# B&R Automation Studio project vibratorControlWithCurrentController (part 5)

#### brdkREST_func.c - Internal functions for library.
```c
#include <brdkREST_func.h>

unsigned short getMethod(brdk_rest_method_typ method) {
	switch(method) {
		case BRDK_REST_GET: return httpMETHOD_GET;
		case BRDK_REST_POST: return httpMETHOD_POST;
		case BRDK_REST_PUT: return httpMETHOD_PUT;
		case BRDK_REST_DELETE: return httpMETHOD_DELETE;
	}
	return httpMETHOD_GET;
}

brdk_rest_method_typ setMethod(unsigned short method) {
	switch(method) {
		case httpMETHOD_GET: return BRDK_REST_GET;
		case httpMETHOD_POST: return BRDK_REST_POST;
		case httpMETHOD_PUT: return BRDK_REST_PUT;
		case httpMETHOD_DELETE: return BRDK_REST_DELETE;
	}
	return BRDK_REST_GET;
}

void setHttpStatus(brdk_rest_response_action_typ status, unsigned long pStr) {
	switch(status) {
		case BRDK_REST_200_OK: brdkStrCpy(pStr, (unsigned long)&"200 OK"); break;
		case BRDK_REST_401_UNAUTHORIZED: brdkStrCpy(pStr, (unsigned long)&"401 Unauthorized"); break;
		case BRDK_REST_403_FORBIDDEN: brdkStrCpy(pStr, (unsigned long)&"403 Forbidden"); break;
		case BRDK_REST_404_NOT_FOUND: brdkStrCpy(pStr, (unsigned long)&"404 Not Found"); break;
		case BRDK_REST_500_INT_SERVER_ERROR: brdkStrCpy(pStr, (unsigned long)&"500 Internal Server Error"); break;
		case BRDK_REST_501_NOT_IMPLEMENTED: brdkStrCpy(pStr, (unsigned long)&"501 Not Implemented"); break;
		case BRDK_REST_503_SRV_UNAVAILABLE: brdkStrCpy(pStr, (unsigned long)&"503 Service Unavailable"); break;
		default: brdkStrCpy(pStr, (unsigned long)&"400 Bad Request"); break;
	}
}

brdk_rest_content_typ findContentType(unsigned long pStr) {
	if(brdkStrSearch(pStr, (unsigned long)&"html") > -1) return BRDK_REST_HTML;
	else if(brdkStrSearch(pStr, (unsigned long)&"plain") > -1) return BRDK_REST_TEXT;
	else if(brdkStrSearch(pStr, (unsigned long)&"json") > -1) return BRDK_REST_JSON;
	else if(brdkStrSearch(pStr, (unsigned long)&"xml") > -1) return BRDK_REST_XML;
	else if(brdkStrSearch(pStr, (unsigned long)&"csv") > -1) return BRDK_REST_CSV;
	else if(brdkStrSearch(pStr, (unsigned long)&"css") > -1) return BRDK_REST_CSS;
	else if(brdkStrSearch(pStr, (unsigned long)&"java") > -1) return BRDK_REST_JAVASCRIPT;
	else if(brdkStrSearch(pStr, (unsigned long)&"jpeg") > -1) return BRDK_REST_JPEG;
	else if(brdkStrSearch(pStr, (unsigned long)&"gzip") > -1) return BRDK_REST_GZIP;
	else if(brdkStrSearch(pStr, (unsigned long)&"zip") > -1) return BRDK_REST_ZIP;
	else if(brdkStrSearch(pStr, (unsigned long)&"png") > -1) return BRDK_REST_PNG;
	else if(brdkStrSearch(pStr, (unsigned long)&"gif") > -1) return BRDK_REST_GIF;
	else if(brdkStrSearch(pStr, (unsigned long)&"bmp") > -1) return BRDK_REST_BMP;
	else if(brdkStrSearch(pStr, (unsigned long)&"jpg") > -1) return BRDK_REST_JPG;
	return BRDK_REST_NONE;
}

void setContentType(unsigned long pDestination, brdk_rest_content_typ type) {
	switch(type) {
		case BRDK_REST_NONE: brdkStrCpy(pDestination,(unsigned long)&""); break;
		case BRDK_REST_HTML: brdkStrCpy(pDestination,(unsigned long)&"text/html"); break;
		case BRDK_REST_TEXT: brdkStrCpy(pDestination,(unsigned long)&"text/plain"); break;
		case BRDK_REST_JSON: brdkStrCpy(pDestination,(unsigned long)&"application/json"); break;
		case BRDK_REST_XML: brdkStrCpy(pDestination,(unsigned long)&"application/xml"); break;
		case BRDK_REST_CSV: brdkStrCpy(pDestination,(unsigned long)&"text/csv"); break;
		case BRDK_REST_CSS: brdkStrCpy(pDestination,(unsigned long)&"text/css"); break;
		case BRDK_REST_JAVASCRIPT: brdkStrCpy(pDestination,(unsigned long)&"text/javascript"); break;
		case BRDK_REST_JPEG: brdkStrCpy(pDestination,(unsigned long)&"image/jpeg"); break;
		case BRDK_REST_GZIP: brdkStrCpy(pDestination,(unsigned long)&"application/gzip"); break;
		case BRDK_REST_ZIP: brdkStrCpy(pDestination,(unsigned long)&"application/zip"); break;
		case BRDK_REST_PNG: brdkStrCpy(pDestination,(unsigned long)&"image/png"); break;
		case BRDK_REST_GIF: brdkStrCpy(pDestination,(unsigned long)&"image/gif"); break;
		case BRDK_REST_BMP: brdkStrCpy(pDestination,(unsigned long)&"image/bmp"); break;
		case BRDK_REST_JPG: brdkStrCpy(pDestination,(unsigned long)&"image/jpg"); break;
	}
}

unsigned char validateServerParams(brdkRESTServer_typ* inst, brdk_rest_server_internal_typ* this) {
	unsigned char i,j,validate = true;
	brdkStrCat((unsigned long)&this->uri, (unsigned long)&"&");
	for(i=0; i <= BRDK_REST_PARAMS_MAX_SIZE; i++) {
		/* try to find in uri */
		if(inst->parameters[i].pKey != 0) {
			validate = false;
			switch(inst->parameters[i].from) {

				case BRDK_REST_PARAMETERS:
					validate = brdkStrSubStrSearch(inst->parameters[i].pValue,(unsigned long)&this->uri,inst->parameters[i].pKey,(unsigned long)&("&"), 1, true);
					break;

				case BRDK_REST_HEADER:
					for(j=0; j <= BRDK_REST_PARAMS_MAX_SIZE; j++) {
						if(brdkStrCmp(inst->parameters[i].pKey, (unsigned long)&this->httpRequestHeader.userLine[j].name) == 0) {
							validate = !brdkStrIsEmpty((unsigned long)&this->httpRequestHeader.userLine[j].value);
							if(validate) {
								brdkStrCpy(inst->parameters[i].pValue, (unsigned long)&this->httpRequestHeader.userLine[j].value);
								break;
							}
						}
					}
					break;

				case BRDK_REST_BODY_JSON:
					switch(inst->parameters[i].datatype) {

						case BRDK_JSON_STRING_TO_STRING: case BRDK_JSON_DINT_TO_STRING: case BRDK_JSON_UDINT_TO_STRING: case BRDK_JSON_BOOL_TO_STRING:
							if(brdkJSONparseToString(inst->pRequestBody, inst->parameters[i].pKey, inst->parameters[i].pValue, inst->parameters[i].datatype, inst->requestBodyMaxLength, 0) > -1) {
								validate = true;
							}
							break;

						default:
							if(brdkJSONparse(inst->pRequestBody, inst->parameters[i].pKey, inst->parameters[i].pValue , inst->parameters[i].datatype, 0) > -1) {
								validate = true;
							}
							break;

					}
					break;

			}
			if(!validate) break;

		}
		else break;
	}
	return validate;
}
```

- CHANGELOG (not shown)

### Library Logical/Libraries/brdkJSON (ANSIC, version 1.00.0) - JSON handling library.
Depends on: brdkSTR

#### brdkJSON.typ - Exported data types
```iecst
TYPE
	brdk_json_find_typ :
		( (*JSON find type.*)
		BRDK_JSON_OBJECT_START := 0, (*JSON object start {.*)
		BRDK_JSON_OBJECT_END := 1, (*JSON object end }.*)
		BRDK_JSON_ARRAY_START := 2, (*JSON array start [.*)
		BRDK_JSON_ARRAY_ELEMENT := 4, (*JSON array element ,.*)
		BRDK_JSON_ARRAY_END := 5, (*JSON array end ].*)
		BRDK_JSON_OBJECT_VALUE := 6, (*JSON value :.*)
		BRDK_JSON_SOURCE_END := 7 (*JSON source end NULL.*)
		);
	brdk_json_dt_typ :
		( (*JSON datatype.*)
		BRDK_JSON_STRING_TO_STRING := 0, (*STRING -> STRING.*)
		BRDK_JSON_STRING_TO_DINT := 1, (*STRING -> DINT.*)
		BRDK_JSON_STRING_TO_UDINT := 2, (*STRING -> UDINT.*)
		BRDK_JSON_STRING_TO_REAL := 3, (*STRING -> REAL.*)
		BRDK_JSON_STRING_TO_BOOL := 4, (*STRING -> BOOL.*)
		BRDK_JSON_DINT_TO_STRING := 5, (*DINT -> STRING.*)
		BRDK_JSON_DINT_TO_DINT := 6, (*DINT -> DINT.*)
		BRDK_JSON_DINT_TO_BOOL := 7, (*DINT -> BOOL.*)
		BRDK_JSON_UDINT_TO_STRING := 8, (*UDINT -> STRING.*)
		BRDK_JSON_UDINT_TO_UDINT := 9, (*UDINT -> UDINT.*)
		BRDK_JSON_UDINT_TO_BOOL := 10, (*UDINT -> BOOL.*)
		BRDK_JSON_BOOL_TO_STRING := 11, (*BOOL -> STRING.*)
		BRDK_JSON_BOOL_TO_DINT := 12, (*BOOL -> DINT.*)
		BRDK_JSON_BOOL_TO_UDINT := 13, (*BOOL -> UDINT.*)
		BRDK_JSON_BOOL_TO_BOOL := 14, (*BOOL -> BOOL.*)
		BRDK_JSON_REAL_TO_REAL := 15, (*REAL -> REAL.*)
		BRDK_JSON_REAL_TO_STRING := 16 (*REAL -> STRING.*)
		);
END_TYPE
```

#### brdkJSON.fun - Exported functions and function blocks
```iecst
FUNCTION brdkJSONfindNext : DINT (*Find a JSON element. $RETURN=position;Position after the found element.*) (*$GROUP=User,$CAT=User,$GROUPICON=User.png,$CATICON=User.png*)
	VAR_INPUT
		pSource : UDINT := 0; (*String pointer to the source string.*)
		find : brdk_json_find_typ := BRDK_JSON_OBJECT_START; (*JSON element to find.*)
		position : UDINT := 0; (*Position in the source string where to starte the search for the element. 0 will start from the beginning.*)
	END_VAR
END_FUNCTION

FUNCTION brdkJSONnextElement : brdk_json_find_typ (*Return the next found JSON element. $RETURN=type;JSON element type.*) (*$GROUP=User,$CAT=User,$GROUPICON=User.png,$CATICON=User.png*)
	VAR_INPUT
		pSource : UDINT := 0; (*String pointer to the source string.*)
		pPposition : UDINT := 0; (*Pointer to the position in the source string where to starte the search for the element. 0 will start from the beginning.*)
	END_VAR
END_FUNCTION

FUNCTION brdkJSONparse : DINT (*Finds a name and value pair in a JSON object. $RETURN=position;Position after the found object. Can be used as position input to search for more values in a source string. See error codes below.*) (*$GROUP=User,$CAT=User,$GROUPICON=User.png,$CATICON=User.png*)
	VAR_INPUT
		pSource : UDINT := 0; (*String pointer to the source string.*)
		pName : UDINT := 0; (*String pointer to the name.*)
		pValue : UDINT := 0; (*String pointer to the value destination.*)
		datatype : brdk_json_dt_typ := BRDK_JSON_DINT_TO_DINT; (*Convert datatype.*)
		position : UDINT := 0; (*Position in the source string where to starte the search for the value. 0 will start from the beginning.*)
	END_VAR
END_FUNCTION

FUNCTION brdkJSONparseArray : DINT (*Finds a name and value pair in a JSON object. $RETURN=position;Position after the found object. Can be used as position input to search for more values in a source string. See error codes below.*) (*$GROUP=User,$CAT=User,$GROUPICON=User.png,$CATICON=User.png*)
	VAR_INPUT
		pSource : UDINT := 0; (*String pointer to the source string.*)
		pName : UDINT := 0; (*String pointer to the name.*)
		pValue : UDINT := 0; (*String pointer to the value destination.*)
		datatype : brdk_json_dt_typ := BRDK_JSON_DINT_TO_DINT; (*Convert datatype.*)
		arraySize : UDINT := 0; (*Maximum size of array (number of elements).*)
		position : UDINT := 0; (*Position in the source string where to starte the search for the value. 0 will start from the beginning.*)
	END_VAR
END_FUNCTION

FUNCTION brdkJSONparseToString : DINT (*Finds a name and value pair in a JSON object. $RETURN=position;Position after the found object. Can be used as position input to search for more values in a source string. See error codes below.*) (*$GROUP=User,$CAT=User,$GROUPICON=User.png,$CATICON=User.png*)
	VAR_INPUT
		pSource : UDINT := 0; (*String pointer to the source string.*)
		pName : UDINT := 0; (*String pointer to the name.*)
		pValue : UDINT := 0; (*String pointer to the value destination.*)
		datatype : brdk_json_dt_typ := BRDK_JSON_STRING_TO_STRING; (*Convert datatype.*)
		size : UDINT := 0; (*Maximum size of the value. Only used when value is a STRING type.*)
		position : UDINT := 0; (*Position in the source string where to starte the search for the value. 0 will start from the beginning.*)
	END_VAR
END_FUNCTION

FUNCTION brdkJSONparseToStringArray : DINT (*Finds a name and value pair in a JSON object. $RETURN=position;Position after the found object. Can be used as position input to search for more values in a source string. See error codes below.*) (*$GROUP=User,$CAT=User,$GROUPICON=User.png,$CATICON=User.png*)
	VAR_INPUT
		pSource : UDINT := 0; (*String pointer to the source string.*)
		pName : UDINT := 0; (*String pointer to the name.*)
		pValue : UDINT := 0; (*String pointer to the value destination.*)
		datatype : brdk_json_dt_typ := BRDK_JSON_STRING_TO_STRING; (*Convert datatype.*)
		size : UDINT := 0; (*Maximum size of the value. Only used when value is a STRING type.*)
		arraySize : UDINT := 0; (*Maximum size of array (number of elements).*)
		position : UDINT := 0; (*Position in the source string where to starte the search for the value. 0 will start from the beginning.*)
	END_VAR
END_FUNCTION

FUNCTION brdkJSONstringify : UDINT (*Add name and value pair to a JSON object. $RETURN=position;Position after the added object. Can be used as position input to search for more values in a source string. See error codes below.*) (*$GROUP=User,$CAT=User,$GROUPICON=User.png,$CATICON=User.png*)
	VAR_INPUT
		pDestination : UDINT := 0; (*String pointer to the destination string.*)
		pName : UDINT := 0; (*String pointer to the name.*)
		pValue : UDINT := 0; (*String pointer to value.*)
		datatype : brdk_json_dt_typ := BRDK_JSON_STRING_TO_STRING; (*Convert datatype.*)
		size : UDINT := 0; (*Maximum size of the destination STRING.*)
		position : UDINT := 0; (*Position in the source string where to starte the search for the value. 0 will start from the beginning or it will search for a }.*)
	END_VAR
END_FUNCTION
```

#### brdkJSONfindNext.c - brdkJSONfindNext implementation.
```c
#include <brdkJSON_func.h>

signed long brdkJSONfindNext(unsigned long pSource, enum brdk_json_find_typ find, unsigned long position) {
	unsigned char findChar;
	switch(find) {
		case BRDK_JSON_OBJECT_START: findChar = BRDK_STR_ASCII_OPEN_BRACE; break;
		case BRDK_JSON_OBJECT_END: findChar = BRDK_STR_ASCII_CLOSE_BRACE; break;
		case BRDK_JSON_ARRAY_START: findChar = BRDK_STR_ASCII_OPEN_BRACKET; break;
		case BRDK_JSON_ARRAY_ELEMENT: findChar = BRDK_STR_ASCII_COMMA; break;
		case BRDK_JSON_ARRAY_END: findChar = BRDK_STR_ASCII_CLOSE_BRACKET; break;
		case BRDK_JSON_OBJECT_VALUE: findChar = BRDK_STR_ASCII_COMMA; break;
		case BRDK_JSON_SOURCE_END: findChar = BRDK_STR_ASCII_NULL; break;
	}
	while(((char*)pSource)[position] != BRDK_STR_ASCII_NULL) {
		if(((char*)pSource)[position++] == findChar) {
			if(((char*)pSource)[position] != BRDK_STR_ASCII_NULL) return position;
			else return -2;
		}
	}
	return -1;
}
```

#### brdkJSONnextElement.c - brdkJSONfindNext implementation.
```c
#include <brdkJSON_func.h>

enum brdk_json_find_typ brdkJSONnextElement(unsigned long pSource, unsigned long pPosition) {
	enum brdk_json_find_typ find = BRDK_JSON_SOURCE_END;
	signed long* pos = (signed long*)pPosition;
	unsigned char run = true;
	while(run) {
		switch(((char*)pSource)[*pos]) {
			case BRDK_STR_ASCII_NULL: find = BRDK_JSON_SOURCE_END; run = false; break;
			case BRDK_STR_ASCII_OPEN_BRACE: find = BRDK_JSON_OBJECT_START; run = false; break;
			case BRDK_STR_ASCII_CLOSE_BRACE: find = BRDK_JSON_OBJECT_END; run = false; break;
			case BRDK_STR_ASCII_OPEN_BRACKET: find = BRDK_JSON_ARRAY_START; run = false; break;
			case BRDK_STR_ASCII_COMMA: find = BRDK_JSON_ARRAY_ELEMENT; run = false; break;
			case BRDK_STR_ASCII_CLOSE_BRACKET: find = BRDK_JSON_ARRAY_END; run = false; break;
			case BRDK_STR_ASCII_COLON: find = BRDK_JSON_OBJECT_VALUE; run = false; break;
			default: *pos += 1; break;
		}

	}
	*pos += 1;
	if(((char*)pSource)[*pos] == BRDK_STR_ASCII_NULL) *pos = -1;
	return find;
}
```

#### brdkJSONparse.c - brdkJSONparse implementation.
```c
#include <brdkJSON_func.h>

signed long brdkJSONparse(unsigned long pSource, unsigned long pName, unsigned long pValue, enum brdk_json_dt_typ datatype, unsigned long position) {
	/* {"test": "1234", "test2": "9876"} */
	/* {"test": 1234, "test": 9876} */
	char str[12], run, quoteCnt = 0;
	signed long i, pos = brdkStrSearch((unsigned long)&(((char*)pSource)[position]), pName);
	if(pos > -1) {
		pos += brdkStrLen(pName) + 2 + position;
		switch(datatype) {

			case BRDK_JSON_DINT_TO_DINT: case BRDK_JSON_STRING_TO_DINT:
			case BRDK_JSON_UDINT_TO_UDINT: case BRDK_JSON_STRING_TO_UDINT:
			case BRDK_JSON_REAL_TO_REAL: case BRDK_JSON_STRING_TO_REAL:
				i = 0;
				run = true;
				while(run) {
					switch(((char*)pSource)[pos]) {
						case BRDK_STR_ASCII_NULL: run = false; pos = -2; break;	/* error null cannot be here */
						case BRDK_STR_ASCII_TAB: case BRDK_STR_ASCII_SPACE: case BRDK_STR_ASCII_COLON: case BRDK_STR_ASCII_CR: case BRDK_STR_ASCII_LF: pos++; break;	/* white space and colon can be ok from beginning */
						case BRDK_STR_ASCII_COMMA: case BRDK_STR_ASCII_CLOSE_BRACE: pos++; run = false; break; /* , or } we are finished */
						case BRDK_STR_ASCII_DOUBLE_QUOTES:
							if(quoteCnt > 1 || datatype == BRDK_JSON_DINT_TO_DINT || datatype == BRDK_JSON_UDINT_TO_UDINT || datatype == BRDK_JSON_REAL_TO_REAL) {
								run = false;
								pos = -3;	/* error illegal character */
							}
							else quoteCnt++;
							pos++;
							break;
						case BRDK_STR_ASCII_HYPHEN:
							if(datatype != BRDK_JSON_DINT_TO_DINT && datatype != BRDK_JSON_STRING_TO_DINT && datatype != BRDK_JSON_REAL_TO_REAL && datatype != BRDK_JSON_STRING_TO_REAL) {
								run = false;
								pos = -3;/* error illegal character */
							}
							else ((char*)str)[i++] = ((char*)pSource)[pos++];
							break;
						case BRDK_STR_ASCII_DOT:
							if(datatype != BRDK_JSON_REAL_TO_REAL && datatype != BRDK_JSON_STRING_TO_REAL) {
								run = false;
								pos = -3;/* error illegal character */
							}
							else ((char*)str)[i++] = ((char*)pSource)[pos++];
							break;
						case BRDK_STR_ASCII_0: case BRDK_STR_ASCII_1: case BRDK_STR_ASCII_2: case BRDK_STR_ASCII_3:
						case BRDK_STR_ASCII_4: case BRDK_STR_ASCII_5: case BRDK_STR_ASCII_6: case BRDK_STR_ASCII_7:
						case BRDK_STR_ASCII_8: case BRDK_STR_ASCII_9:
							((char*)str)[i++] = ((char*)pSource)[pos++];
							break;
						default: run = false; pos = -3; break;	/* error illegal character */
					}
				}
				if(pos > -1) {
					((char*)str)[i] = BRDK_STR_ASCII_NULL;
					setValue(datatype, pValue, (unsigned long)&str);
				}
				break;

			case BRDK_JSON_BOOL_TO_BOOL: case BRDK_JSON_STRING_TO_BOOL: case BRDK_JSON_UDINT_TO_BOOL:
			case BRDK_JSON_DINT_TO_BOOL: case BRDK_JSON_BOOL_TO_DINT: case BRDK_JSON_BOOL_TO_UDINT:
				i = 0;
				run = true;
				while(run) {
					switch(((char*)pSource)[pos]) {
						case BRDK_STR_ASCII_NULL: run = false; pos = -2; break;	/* error null cannot be here */
						case BRDK_STR_ASCII_TAB: case BRDK_STR_ASCII_CR: case BRDK_STR_ASCII_LF: case BRDK_STR_ASCII_SPACE: case BRDK_STR_ASCII_COLON: pos++; break;	/* white space can be ok from beginning */
						case BRDK_STR_ASCII_DOUBLE_QUOTES:
							if(quoteCnt > 1 || datatype == BRDK_JSON_BOOL_TO_BOOL || datatype == BRDK_JSON_DINT_TO_BOOL ||
								datatype == BRDK_JSON_UDINT_TO_BOOL || datatype == BRDK_JSON_BOOL_TO_DINT || datatype == BRDK_JSON_BOOL_TO_UDINT) {
								run = false;
								pos = -3;	/* error illegal character */
							}
							else quoteCnt++;
							pos++;
							break;
						case BRDK_STR_ASCII_COMMA: case BRDK_STR_ASCII_CLOSE_BRACE: pos++; run = false; break; /* , or } we are finished */
						case BRDK_STR_ASCII_t: case BRDK_STR_ASCII_r: case BRDK_STR_ASCII_u: case BRDK_STR_ASCII_e:
						case BRDK_STR_ASCII_f: case BRDK_STR_ASCII_a: case BRDK_STR_ASCII_l: case BRDK_STR_ASCII_s:
							if(datatype != BRDK_JSON_UDINT_TO_BOOL && datatype != BRDK_JSON_DINT_TO_BOOL) ((char*)str)[i++] = ((char*)pSource)[pos++];
							else {
								run = false;
								pos = -3;	/* error illegal character */
							}
							break;

						case BRDK_STR_ASCII_0: case BRDK_STR_ASCII_1:
							((char*)str)[i++] = ((char*)pSource)[pos++];
							break;
						default: run = false; pos = -3; break;	/* error illegal character */
					}
				}
				if(pos > -1) {
					((char*)str)[i] = BRDK_STR_ASCII_NULL;
					if(datatype == BRDK_JSON_BOOL_TO_DINT) {
						signed long* tmpVal = ((signed long*)pValue);
						if(brdkStrCmp((unsigned long)&str, (unsigned long)&"true") == 0) *tmpVal = true;
						else if(brdkStrCmp((unsigned long)&str, (unsigned long)&"false") == 0) *tmpVal = false;
						else pos = -3; break;	/* error illegal character */
					}
					else if(datatype == BRDK_JSON_BOOL_TO_UDINT) {
						unsigned long* tmpVal = ((unsigned long*)pValue);
						if(brdkStrCmp((unsigned long)&str, (unsigned long)&"true") == 0) *tmpVal = true;
						else if(brdkStrCmp((unsigned long)&str, (unsigned long)&"false") == 0) *tmpVal = false;
						else pos = -3; break;	/* error illegal character */
					}
					else {
						char* tmpVal = ((char*)pValue);
						if(brdkStrCmp((unsigned long)&str, (unsigned long)&"true") == 0) *tmpVal = true;
						else if(brdkStrCmp((unsigned long)&str, (unsigned long)&"1") == 0) *tmpVal = true;
						else if(brdkStrCmp((unsigned long)&str, (unsigned long)&"false") == 0) *tmpVal = false;
						else if(brdkStrCmp((unsigned long)&str, (unsigned long)&"0") == 0) *tmpVal = false;
						else pos = -3; break;	/* error illegal character */
					}
				}
				break;

			default:
				run = false;
				pos = -4;	/* error not supported in this function */
				break;

		}
	}
	return pos;
}
```

#### brdkJSONparseArray.c - brdkJSONparseArray implementation.
```c
#include <brdkJSON_func.h>

signed long brdkJSONparseArray(unsigned long pSource, unsigned long pName, unsigned long pValue, enum brdk_json_dt_typ datatype, unsigned long arraySize, unsigned long position) {
	/* {"test": "1234", "test2": "9876"} */
	/* {"test": 1234, "test": 9876} */
	char str[12], run, quoteCnt = 0, bracketOpen = false;
	signed long i, index = 0, pos = 0;
	if(pName != 0) pos = brdkStrSearch((unsigned long)&(((char*)pSource)[position]), pName);
	if(pos > -1) {
		if(pName != 0) pos += brdkStrLen(pName) + 2 + position;
		switch(datatype) {

			case BRDK_JSON_DINT_TO_DINT: case BRDK_JSON_STRING_TO_DINT:
			case BRDK_JSON_UDINT_TO_UDINT: case BRDK_JSON_STRING_TO_UDINT:
			case BRDK_JSON_REAL_TO_REAL: case BRDK_JSON_STRING_TO_REAL:
				i = 0;
				run = true;
				while(run) {
					switch(((char*)pSource)[pos]) {
						case BRDK_STR_ASCII_NULL: run = false; pos = -2; break;	/* error null cannot be here */
						case BRDK_STR_ASCII_TAB: case BRDK_STR_ASCII_CR: case BRDK_STR_ASCII_LF: case BRDK_STR_ASCII_SPACE: case BRDK_STR_ASCII_COLON: pos++; break;	/* white space and colon can be ok from beginning */
						case BRDK_STR_ASCII_OPEN_BRACKET:
							bracketOpen = true;
							pos++;
							break;
						case BRDK_STR_ASCII_CLOSE_BRACKET:
							bracketOpen = false;
							pos++;
							if(pName == 0) {
								((char*)str)[i] = BRDK_STR_ASCII_NULL;
								setValue(datatype, pValue, (unsigned long)&str);
								pValue += 4;
								for(;index < arraySize; index++) {
									setValue(datatype, pValue, (unsigned long)&"");
									pValue += 4;
								}
								run = false;
							}
							break;
						case BRDK_STR_ASCII_CLOSE_BRACE:
							pos++;
							((char*)str)[i] = BRDK_STR_ASCII_NULL;
							setValue(datatype, pValue, (unsigned long)&str);
							pValue += 4;
							for(;index < arraySize; index++) {
								setValue(datatype, pValue, (unsigned long)&"");
								pValue += 4;
							}
							run = false;
							break; /* ] we are finished */
						case BRDK_STR_ASCII_COMMA:
							pos++;
							((char*)str)[i] = BRDK_STR_ASCII_NULL;
							setValue(datatype, pValue, (unsigned long)&str);
							pValue += 4;
							if(!bracketOpen) { /* , we are finished */
								for(;index < arraySize; index++) {
									setValue(datatype, pValue, (unsigned long)&"");
									pValue += 4;
								}
								run = false;
							}
							else {	/* bracket still open -> next element in array */
								index++;
								if(index < arraySize) {
									quoteCnt = 0;
									i = 0;
								}
								else {
									run = false;
									pos = -6;	/* array size too small */
								}
							}
							break;
						case BRDK_STR_ASCII_DOUBLE_QUOTES:
							if(quoteCnt > 1 || datatype == BRDK_JSON_DINT_TO_DINT || datatype == BRDK_JSON_UDINT_TO_UDINT || datatype == BRDK_JSON_REAL_TO_REAL) {
								run = false;
								pos = -3;	/* error illegal character */
							}
							else quoteCnt++;
							pos++;
							break;
						case BRDK_STR_ASCII_HYPHEN:
							if(datatype != BRDK_JSON_DINT_TO_DINT && datatype != BRDK_JSON_STRING_TO_DINT && datatype != BRDK_JSON_REAL_TO_REAL && datatype != BRDK_JSON_STRING_TO_REAL) {
								run = false;
								pos = -3;/* error illegal character */
							}
							else ((char*)str)[i++] = ((char*)pSource)[pos++];
							break;
						case BRDK_STR_ASCII_DOT:
							if(datatype != BRDK_JSON_REAL_TO_REAL && datatype != BRDK_JSON_STRING_TO_REAL) {
								run = false;
								pos = -3;/* error illegal character */
							}
							else ((char*)str)[i++] = ((char*)pSource)[pos++];
							break;
						case BRDK_STR_ASCII_0: case BRDK_STR_ASCII_1: case BRDK_STR_ASCII_2: case BRDK_STR_ASCII_3:
						case BRDK_STR_ASCII_4: case BRDK_STR_ASCII_5: case BRDK_STR_ASCII_6: case BRDK_STR_ASCII_7:
						case BRDK_STR_ASCII_8: case BRDK_STR_ASCII_9:
							((char*)str)[i++] = ((char*)pSource)[pos++];
							break;
						default: run = false; pos = -3; break;	/* error illegal character */
					}
				}
				break;

			case BRDK_JSON_BOOL_TO_BOOL: case BRDK_JSON_STRING_TO_BOOL: case BRDK_JSON_DINT_TO_BOOL:
			case BRDK_JSON_UDINT_TO_BOOL: case BRDK_JSON_BOOL_TO_DINT: case BRDK_JSON_BOOL_TO_UDINT:
				i = 0;
				run = true;
				while(run) {
					switch(((char*)pSource)[pos]) {
						case BRDK_STR_ASCII_NULL: run = false; pos = -2; break;	/* error null cannot be here */
						case BRDK_STR_ASCII_TAB: case BRDK_STR_ASCII_CR: case BRDK_STR_ASCII_LF: case BRDK_STR_ASCII_SPACE: case BRDK_STR_ASCII_COLON: pos++; break;	/* white space can be ok from beginning */
						case BRDK_STR_ASCII_DOUBLE_QUOTES:
							if(quoteCnt > 1 || datatype == BRDK_JSON_BOOL_TO_BOOL || datatype == BRDK_JSON_DINT_TO_BOOL ||
								datatype == BRDK_JSON_UDINT_TO_BOOL || datatype == BRDK_JSON_BOOL_TO_DINT || datatype == BRDK_JSON_BOOL_TO_UDINT) {
								run = false;
								pos = -3;	/* error illegal character */
							}
							else quoteCnt++;
							pos++;
							break;
						case BRDK_STR_ASCII_OPEN_BRACKET:
							bracketOpen = true;
							pos++;
							break;
						case BRDK_STR_ASCII_CLOSE_BRACKET:
							bracketOpen = false;
							pos++;
							if(pName == 0) {
								((char*)str)[i] = BRDK_STR_ASCII_NULL;
								if(setValue(datatype, pValue, (unsigned long)&str) != 0) {
									pos = -3;
									run = false;
									break;
								}
								pValue += getSize(datatype);
								for(;index < arraySize; index++) {
									if(setValue(datatype, pValue, (unsigned long)&"0") != 0) {
										pos = -3;
										run = false;
										break;
									}
									pValue += getSize(datatype);
								}
								run = false;
							}
							break; /* } we are finished */
						case BRDK_STR_ASCII_COMMA:
							pos++;
							((char*)str)[i] = BRDK_STR_ASCII_NULL;
							if(setValue(datatype, pValue, (unsigned long)&str) != 0) {
								pos = -3;
								run = false;
							}
							pValue += getSize(datatype);
							if(!bracketOpen) { /* , we are finished */
								for(;index < arraySize; index++) {
									if(setValue(datatype, pValue, (unsigned long)&"0") != 0) {
										pos = -3;
										run = false;
										break;
									}
									pValue += getSize(datatype);
								}
								run = false;
							}
							else {	/* bracket still open -> next element in array */
								index++;
								if(index < arraySize) {
									quoteCnt = 0;
									i = 0;
								}
								else {
									run = false;
									pos = -6;	/* array size too small */
								}
							}
							break;
						case BRDK_STR_ASCII_CLOSE_BRACE:
							pos++;
							((char*)str)[i] = BRDK_STR_ASCII_NULL;
							if(setValue(datatype, pValue, (unsigned long)&str) != 0) {
								pos = -3;
								run = false;
							}
							pValue += getSize(datatype);
							for(;index < arraySize; index++) {
								if(setValue(datatype, pValue, (unsigned long)&"0") != 0) {
									pos = -3;
									run = false;
								}
								pValue += getSize(datatype);
							}
							run = false;
							break; /* } we are finished */
						case BRDK_STR_ASCII_t: case BRDK_STR_ASCII_r: case BRDK_STR_ASCII_u: case BRDK_STR_ASCII_e:
						case BRDK_STR_ASCII_f: case BRDK_STR_ASCII_a: case BRDK_STR_ASCII_l: case BRDK_STR_ASCII_s:
							if(datatype != BRDK_JSON_UDINT_TO_BOOL && datatype != BRDK_JSON_DINT_TO_BOOL) ((char*)str)[i++] = ((char*)pSource)[pos++];
							else {
								run = false;
								pos = -3;	/* error illegal character */
							}
							break;

						case BRDK_STR_ASCII_0: case BRDK_STR_ASCII_1:
							((char*)str)[i++] = ((char*)pSource)[pos++];
							break;
						default: run = false; pos = -3; break;	/* error illegal character */
					}
				}
				break;

			default:
				run = false;
				pos = -4;	/* error not supported in this function */
				break;

		}
	}
	return pos;
}
```

#### brdkJSONparseToString.c - brdkJSONparseToString implementation.
```c
#include <brdkJSON_func.h>

signed long brdkJSONparseToString(unsigned long pSource, unsigned long pName, unsigned long pValue, enum brdk_json_dt_typ datatype, unsigned long size, unsigned long position) {
	/* {"test": "1234", "test2": "9876"} */
	/* {"test": 1234, "test": 9876} */
	char run, quoteCnt = 0;
	signed long i, pos = brdkStrSearch((unsigned long)&(((char*)pSource)[position]), pName);
	if(pos > -1) {
		pos += brdkStrLen(pName) + 2 + position;
		switch(datatype) {

			case BRDK_JSON_STRING_TO_STRING: case BRDK_JSON_DINT_TO_STRING: case BRDK_JSON_UDINT_TO_STRING: case BRDK_JSON_BOOL_TO_STRING: case BRDK_JSON_REAL_TO_STRING:
				i = 0;
				run = true;
				char bckslash = false;
				while(run) {
					/* find first double quote */
					switch(((char*)pSource)[pos]) {
						case BRDK_STR_ASCII_NULL: run = false; pos = -2; break;	/* error null cannot be here */
						case BRDK_STR_ASCII_TAB: case BRDK_STR_ASCII_CR: case BRDK_STR_ASCII_LF: pos++; break;
						case BRDK_STR_ASCII_COMMA: case BRDK_STR_ASCII_CLOSE_BRACE:
							if(quoteCnt < 2 && datatype == BRDK_JSON_STRING_TO_STRING) {
								if(i < size) ((char*)pValue)[i++] = ((char*)pSource)[pos++];
								else {
									run = false;
									pos = -5;	/* error string size too small */
								}
							}
							else {
								pos++;
								run = false;
								((char*)pValue)[i] = BRDK_STR_ASCII_NULL;
							}
							break;
						case BRDK_STR_ASCII_DOT:
							if(datatype == BRDK_JSON_REAL_TO_STRING || datatype == BRDK_JSON_STRING_TO_STRING) {
								if(i < size) ((char*)pValue)[i++] = ((char*)pSource)[pos++];
								else {
									run = false;
									pos = -5;	/* error string size too small */
								}
							}
							else {
								run = false;
								pos = -3;	/* error illegal character */
							}
							break;
						case BRDK_STR_ASCII_DOUBLE_QUOTES:
							if(datatype == BRDK_JSON_STRING_TO_STRING) {
								if(!bckslash) {
									if(quoteCnt > 1) {
										run = false;
										pos = -3;	/* error illegal character */
									}
									else quoteCnt++;
								}
								else bckslash = false;
								pos++;
							}
							else {
								run = false;
								pos = -3;	/* error illegal character */
							}
							break;
						case BRDK_STR_ASCII_HYPHEN:
							if(datatype == BRDK_JSON_DINT_TO_STRING || datatype == BRDK_JSON_STRING_TO_STRING || datatype == BRDK_JSON_REAL_TO_STRING) {
								if(i < size) ((char*)pValue)[i++] = ((char*)pSource)[pos++];
								else {
									run = false;
									pos = -5;	/* error string size too small */
								}
							}
							else {
								run = false;
								pos = -3;/* error illegal character */
							}
							break;
						case BRDK_STR_ASCII_BACK_SLASH:
							if(datatype == BRDK_JSON_STRING_TO_STRING) {
								if(!bckslash) bckslash = true;
								else {
									if(i < size) {
										((char*)pValue)[i++] = ((char*)pSource)[pos];
										bckslash = false;
									}
									else {
										run = false;
										pos = -5;	/* error string size too small */
									}
								}
								if(run) pos++;
							}
							else {
								run = false;
								pos = -3;	/* error illegal character */
							}
							break;
						case BRDK_STR_ASCII_SPACE: case BRDK_STR_ASCII_COLON:
							if(quoteCnt == 1) {
								if(i < size) ((char*)pValue)[i++] = ((char*)pSource)[pos];
								else {
									run = false;
									pos = -5;	/* error string size too small */
								}
							}
							if(run) pos++;
							break;
						default:
							if(datatype == BRDK_JSON_STRING_TO_STRING) {
								if(quoteCnt > 0) {
									if(i < size) ((char*)pValue)[i++] = ((char*)pSource)[pos++];
									else {
										run = false;
										pos = -5;	/* error string size too small */
									}
								}
								else {
									run = false;
									pos = -3;	/* error illegal character */
								}
							}
							else if(datatype == BRDK_JSON_DINT_TO_STRING || datatype == BRDK_JSON_UDINT_TO_STRING || datatype == BRDK_JSON_REAL_TO_STRING) {
								switch(((char*)pSource)[pos]) {
									case BRDK_STR_ASCII_0: case BRDK_STR_ASCII_1: case BRDK_STR_ASCII_2: case BRDK_STR_ASCII_3:
									case BRDK_STR_ASCII_4: case BRDK_STR_ASCII_5: case BRDK_STR_ASCII_6: case BRDK_STR_ASCII_7:
									case BRDK_STR_ASCII_8: case BRDK_STR_ASCII_9:
										if(i < size) ((char*)pValue)[i++] = ((char*)pSource)[pos++];
										else {
											run = false;
											pos = -5;	/* error string size too small */
										}
										break;

									default:
										run = false;
										pos = -3;	/* error illegal character */
										break;
								}
							}
							else if(datatype == BRDK_JSON_BOOL_TO_STRING) {
								switch(((char*)pSource)[pos]) {
										case BRDK_STR_ASCII_t: case BRDK_STR_ASCII_r: case BRDK_STR_ASCII_u: case BRDK_STR_ASCII_e:
										case BRDK_STR_ASCII_f: case BRDK_STR_ASCII_a: case BRDK_STR_ASCII_l: case BRDK_STR_ASCII_s:
										if(i < size) ((char*)pValue)[i++] = ((char*)pSource)[pos++];
										else {
											run = false;
											pos = -5;	/* error string size too small */
										}
										break;

									default:
										run = false;
										pos = -3;	/* error illegal character */
										break;
								}
							}
							break;
					}
				}
				break;

			default:
				run = false;
				pos = -4;	/* error not supported in this function */
				break;
		}
	}
	return pos;
}
```

#### brdkJSONparseToStringArray.c - brdkJSONparseToStringArray implementation.
```c
#include <brdkJSON_func.h>

signed long brdkJSONparseToStringArray(unsigned long pSource, unsigned long pName, unsigned long pValue, enum brdk_json_dt_typ datatype, unsigned long size, unsigned long arraySize, unsigned long position) {
	char run, quoteCnt = 0, bracketOpen = false;
	signed long i, index = 0, pos = 0;
	if(pName != 0) pos = brdkStrSearch((unsigned long)&(((char*)pSource)[position]), pName);
	if(pos > -1) {
		if(pName != 0) pos += brdkStrLen(pName) + 2 + position;
		switch(datatype) {

			case BRDK_JSON_STRING_TO_STRING: case BRDK_JSON_DINT_TO_STRING: case BRDK_JSON_UDINT_TO_STRING: case BRDK_JSON_BOOL_TO_STRING: case BRDK_JSON_REAL_TO_STRING:
				i = 0;
				run = true;
				char bckslash = false;
				while(run) {
					/* find the first square bracket */
					switch(((char*)pSource)[pos]) {
						case BRDK_STR_ASCII_NULL: run = false; pos = -2; break;	/* error null cannot be here */
						case BRDK_STR_ASCII_TAB: case BRDK_STR_ASCII_CR: case BRDK_STR_ASCII_LF: pos++; break;
						case BRDK_STR_ASCII_CLOSE_BRACKET:
							if(bracketOpen && quoteCnt == 1 && datatype == BRDK_JSON_STRING_TO_STRING) {
								if(i < size) ((char*)pValue)[i++] = ((char*)pSource)[pos];
								else {
									run = false;
									pos = -5;	/* error string size too small */
								}
							}
							else {
								bracketOpen = false;
								if(pName != 0) {
									if(run) pos++;	/* pName == 0 is allowed for e.g. [1,2,3] */
								}
								else {
									((char*)pValue)[i] = BRDK_STR_ASCII_NULL;
									i = 0;
									for(;index < arraySize; index++) {
										pValue += size;
										((char*)pValue)[i] = BRDK_STR_ASCII_NULL;
									}
									pos++;
									run = false;
								}
							}
							break;
						case BRDK_STR_ASCII_COMMA:
							if(quoteCnt < 2 && datatype == BRDK_JSON_STRING_TO_STRING) {
								if(!bracketOpen) {
								 	i = 0;
									for(;index < arraySize; index++) {
										pValue += size;
										((char*)pValue)[i] = BRDK_STR_ASCII_NULL;
									}
									run = false;
								}
								else {
									if(i < size) ((char*)pValue)[i++] = ((char*)pSource)[pos++];
									else {
										run = false;
										pos = -5;	/* error string size too small */
									}
								}
							}
							else {
								((char*)pValue)[i] = BRDK_STR_ASCII_NULL;
								pos++;
								/* bracket is closed -> comma after array element -> we are finished */
								if(!bracketOpen) {
								 	i = 0;
									for(;index < arraySize; index++) {
										pValue += size;
										((char*)pValue)[i] = BRDK_STR_ASCII_NULL;
									}
									run = false;
								}
								else {	/* bracket still open -> next element in array */
									index++;
									if(index < arraySize) {
										pValue += size;
										quoteCnt = 0;
										i = 0;
									}
									else {
										run = false;
										pos = -6;	/* array size too small */
									}
								}
							}
							break;
						case BRDK_STR_ASCII_CLOSE_BRACE:
							if(quoteCnt == 1 && datatype == BRDK_JSON_STRING_TO_STRING)
								if(i < size) ((char*)pValue)[i++] = ((char*)pSource)[pos++];
								else {
									run = false;
									pos = -5;	/* error string size too small */
								}
							else {
								if(datatype != BRDK_JSON_STRING_TO_STRING) ((char*)pValue)[i] = BRDK_STR_ASCII_NULL;
								i = 0;
								for(;index < arraySize; index++) {
									pValue += size;
									((char*)pValue)[i] = BRDK_STR_ASCII_NULL;
								}
								pos++;
								run = false;
							}
							break;
						case BRDK_STR_ASCII_DOUBLE_QUOTES:
							if(datatype == BRDK_JSON_STRING_TO_STRING) {
								if(!bckslash) {
									if(quoteCnt > 1) {
										run = false;
										pos = -3;	/* error illegal character */
									}
									else quoteCnt++;
								}
								else bckslash = false;
								pos++;
							}
							else {
								run = false;
								pos = -3;	/* error illegal character */
							}
							break;
						case BRDK_STR_ASCII_HYPHEN:
							if(datatype == BRDK_JSON_DINT_TO_STRING || datatype == BRDK_JSON_STRING_TO_STRING || datatype == BRDK_JSON_REAL_TO_STRING) {
								if(i < size) ((char*)pValue)[i++] = ((char*)pSource)[pos++];
								else {
									run = false;
									pos = -5;	/* error string size too small */
								}
							}
							else {
								run = false;
								pos = -3;/* error illegal character */
							}
							break;
						case BRDK_STR_ASCII_DOT:
							if(datatype == BRDK_JSON_REAL_TO_STRING || datatype == BRDK_JSON_STRING_TO_STRING) {
								if(i < size) ((char*)pValue)[i++] = ((char*)pSource)[pos++];
								else {
									run = false;
									pos = -5;	/* error string size too small */
								}
							}
							else {
								run = false;
								pos = -3;	/* error illegal character */
							}
							break;
						case BRDK_STR_ASCII_BACK_SLASH:
							if(datatype == BRDK_JSON_STRING_TO_STRING) {
								if(!bckslash) bckslash = true;
								else {
									if(i < size) {
										((char*)pValue)[i++] = ((char*)pSource)[pos];
										bckslash = false;
									}
									else {
										run = false;
										pos = -5;	/* error string size too small */
									}
								}
								if(run) pos++;
							}
							else {
								run = false;
								pos = -3;	/* error illegal character */
							}
							break;
						case BRDK_STR_ASCII_SPACE: case BRDK_STR_ASCII_COLON:
							if(quoteCnt == 1) {
								if(i < size) ((char*)pValue)[i++] = ((char*)pSource)[pos];
								else {
									run = false;
									pos = -5;	/* error string size too small */
								}
							}
							if(run) pos++;
							break;
						case BRDK_STR_ASCII_OPEN_BRACKET:
							bracketOpen = true;
							if(quoteCnt > 0) {
								if(i < size) ((char*)pValue)[i++] = ((char*)pSource)[pos];
								else {
									run = false;
									pos = -5;	/* error string size too small */
								}
							}
							if(run) pos++;
							break;
						default:
							if(datatype == BRDK_JSON_STRING_TO_STRING) {
								if(quoteCnt > 0) {
									if(i < size) ((char*)pValue)[i++] = ((char*)pSource)[pos++];
									else {
										run = false;
										pos = -5;	/* error string size too small */
									}
								}
								else {
									run = false;
									pos = -3;	/* error illegal character */
								}
							}
							else if(datatype == BRDK_JSON_DINT_TO_STRING || datatype == BRDK_JSON_UDINT_TO_STRING || datatype == BRDK_JSON_REAL_TO_STRING) {
								switch(((char*)pSource)[pos]) {
									case BRDK_STR_ASCII_0: case BRDK_STR_ASCII_1: case BRDK_STR_ASCII_2: case BRDK_STR_ASCII_3:
									case BRDK_STR_ASCII_4: case BRDK_STR_ASCII_5: case BRDK_STR_ASCII_6: case BRDK_STR_ASCII_7:
									case BRDK_STR_ASCII_8: case BRDK_STR_ASCII_9:
										if(i < size) ((char*)pValue)[i++] = ((char*)pSource)[pos++];
										else {
											run = false;
											pos = -5;	/* error string size too small */
										}
										break;

									default:
										run = false;
										pos = -3;	/* error illegal character */
										break;
								}
							}
							else if(datatype == BRDK_JSON_BOOL_TO_STRING) {
								switch(((char*)pSource)[pos]) {
										case BRDK_STR_ASCII_t: case BRDK_STR_ASCII_r: case BRDK_STR_ASCII_u: case BRDK_STR_ASCII_e:
										case BRDK_STR_ASCII_f: case BRDK_STR_ASCII_a: case BRDK_STR_ASCII_l: case BRDK_STR_ASCII_s:
										if(i < size) ((char*)pValue)[i++] = ((char*)pSource)[pos++];
										else {
											run = false;
											pos = -5;	/* error string size too small */
										}
										break;

									default:
										run = false;
										pos = -3;	/* error illegal character */
										break;
								}
							}
							break;
					}
				}
				break;

			default:
				run = false;
				pos = -4;	/* error not supported in this function */
				break;
		}
	}
	return pos;
}
```

#### brdkJSONstringify.c - brdkJSONstringify implementation.
```c
#include <brdkJSON_func.h>

unsigned long brdkJSONstringify(unsigned long pDestination, unsigned long pName, unsigned long pValue, enum brdk_json_dt_typ datatype, unsigned long size, unsigned long position) {
	unsigned long i = 0;
	if(position == 0) {
		while(((char*)pDestination)[position] != BRDK_STR_ASCII_NULL && ((char*)pDestination)[position] != BRDK_STR_ASCII_CLOSE_BRACE) {
			position++;
		}
	}
	if(position < (size-2)) {
		if(position != 0) ((char*)pDestination)[position++] = BRDK_STR_ASCII_COMMA;		/* property before, add comma */
		else ((char*)pDestination)[position++] = BRDK_STR_ASCII_OPEN_BRACE;				/* first property, add open brace */
		((char*)pDestination)[position++] = BRDK_STR_ASCII_DOUBLE_QUOTES;				/* add double quote for name */
	}
	else return -5;

	while(((char*)pName)[i] != BRDK_STR_ASCII_NULL) {
		if(position < size) ((char*)pDestination)[position++] = ((char*)pName)[i++];	/* add name */
		else return -5;
	}
	if(position < (size-2)) {
		((char*)pDestination)[position++] = BRDK_STR_ASCII_DOUBLE_QUOTES;				/* add last double quote of name */
		((char*)pDestination)[position++] = BRDK_STR_ASCII_COLON;						/* add colon before value */
	}
	else return -5;

	switch(datatype) {

		case BRDK_JSON_STRING_TO_STRING:
			if(position < size) ((char*)pDestination)[position++] = BRDK_STR_ASCII_DOUBLE_QUOTES;
			else return -5;
			i = 0;
			while(((char*)pValue)[i] != BRDK_STR_ASCII_NULL) {
				if(position < size) ((char*)pDestination)[position++] = ((char*)pValue)[i++];
				else return -5;
			}
			if(position < size) ((char*)pDestination)[position++] = BRDK_STR_ASCII_DOUBLE_QUOTES;
			else return -5;
			break;

		case BRDK_JSON_STRING_TO_UDINT: case BRDK_JSON_STRING_TO_DINT: case BRDK_JSON_STRING_TO_REAL:
			i = 0;
			while(((char*)pValue)[i] != BRDK_STR_ASCII_NULL) {
				if(position < size) ((char*)pDestination)[position++] = ((char*)pValue)[i++];
				else return -5;
			}
			break;

		case BRDK_JSON_STRING_TO_BOOL:
			if(position < (size-5)) {
				if(brdkStrCmp(pValue,(unsigned long)&"false") == 0 || brdkStrCmp(pValue,(unsigned long)&"0") == 0) {
					position = appendBOOL(false, pDestination, position, size);
				}
				else if(brdkStrCmp(pValue,(unsigned long)&"true") == 0 || brdkStrCmp(pValue,(unsigned long)&"1") == 0) {
					position = appendBOOL(true, pDestination, position, size);
				}
			}
			else return -5;
			break;

		case BRDK_JSON_DINT_TO_STRING:
			if(position < (size-13)) {	/* max. size of DINT + hypen + 2 x double quotes */
				((char*)pDestination)[position++] = BRDK_STR_ASCII_DOUBLE_QUOTES;
				signed long* tmpVal = ((signed long*)pValue);
				brdkStrAppendDintToA(*tmpVal,pDestination,BRDK_STR_CONVERT_DECIMAL,position);
				position += brdkStrDintLen(*tmpVal);
				((char*)pDestination)[position++] = BRDK_STR_ASCII_DOUBLE_QUOTES;
			}
			else return -5;
			break;

		case BRDK_JSON_DINT_TO_DINT:
			if(position < (size-11)) {	/* max. size of DINT + hypen */
				signed long* tmpVal = ((signed long*)pValue);
				brdkStrAppendDintToA(*tmpVal,pDestination,BRDK_STR_CONVERT_DECIMAL,position);
				position += brdkStrDintLen(*tmpVal);
			}
			else return -5;
			break;

		case BRDK_JSON_DINT_TO_BOOL:
			if(position < (size-6)) {	/* max. size of false */
				signed long* tmpVal = ((signed long*)pValue);
				if(!*tmpVal) position = appendBOOL(false, pDestination, position, size);
				else position = appendBOOL(true, pDestination, position, size);
			}
			else return -5;
			break;

		case BRDK_JSON_UDINT_TO_STRING:
			if(position < (size-12)) {	/* max. size of UDINT + 2 x double quotes */
				((char*)pDestination)[position++] = BRDK_STR_ASCII_DOUBLE_QUOTES;
				unsigned long* tmpVal = ((unsigned long*)pValue);
				brdkStrAppendUdintToA(*tmpVal,pDestination,BRDK_STR_CONVERT_DECIMAL,position);
				position += brdkStrUdintLen(*tmpVal);
				((char*)pDestination)[position++] = BRDK_STR_ASCII_DOUBLE_QUOTES;
			}
			else return -5;
			break;

		case BRDK_JSON_UDINT_TO_UDINT:
			if(position < (size-10)) {	/* max. size of UDINT */
				unsigned long* tmpVal = ((unsigned long*)pValue);
				brdkStrAppendUdintToA(*tmpVal,pDestination,BRDK_STR_CONVERT_DECIMAL,position);
				position += brdkStrUdintLen(*tmpVal);
			}
			else return -5;
			break;

		case BRDK_JSON_UDINT_TO_BOOL:
			if(position < (size-6)) {	/* max. size of false */
				unsigned long* tmpVal = ((unsigned long*)pValue);
				if(!*tmpVal) position = appendBOOL(false, pDestination, position, size);
				else position = appendBOOL(true, pDestination, position, size);
			}
			else return -5;
			break;

		case BRDK_JSON_BOOL_TO_STRING:
			if(position < (size-8)) {	/* max. size of false + 2 x diuble quotes */
				((char*)pDestination)[position++] = BRDK_STR_ASCII_DOUBLE_QUOTES;
				char* tmpVal = ((char*)pValue);
				if(!*tmpVal) position = appendBOOL(false, pDestination, position, size);
				else position = appendBOOL(true, pDestination, position, size);
				((char*)pDestination)[position++] = BRDK_STR_ASCII_DOUBLE_QUOTES;
			}
			else return -5;
			break;

		case BRDK_JSON_BOOL_TO_UDINT: case BRDK_JSON_BOOL_TO_DINT:
			if(position < size) {	/* max. size of 1 */
				char* tmpVal = ((char*)pValue);
				if(!*tmpVal) ((char*)pDestination)[position++] = BRDK_STR_ASCII_0;
				else ((char*)pDestination)[position++] = BRDK_STR_ASCII_1;
			}
			else return -5;
			break;

		case BRDK_JSON_BOOL_TO_BOOL:
			if(position < (size-6)) {	/* max. size of false */
				char* tmpVal = ((char*)pValue);
				if(!*tmpVal) position = appendBOOL(false, pDestination, position, size);
				else position = appendBOOL(true, pDestination, position, size);
			}
			else return -5;
			break;

		default:
			return -4;	/* error not supported in this function */
			break;

	}
	if(position < (size-2)) {
		((char*)pDestination)[position] = BRDK_STR_ASCII_CLOSE_BRACE;
		((char*)pDestination)[position+1] = BRDK_STR_ASCII_NULL;
	}
	else return -5;
	return position;
}
```

- CHANGELOG (not shown)

#### brdkJSON_func.h - Header for internal functions for library.
```c
#ifndef BRDK_JSON_FUNCS
#define BRDK_JSON_FUNCS 1

#include <brdkJSON.h>
#include <bur/plctypes.h>

#ifdef __cplusplus
	extern "C"
	{
#endif

#ifdef __cplusplus
	};
#endif

#define false 0
#define true 1
#define NULL 0

unsigned long appendBOOL(char value, unsigned long pDestination, unsigned long position, unsigned long size);
unsigned long setValue(enum brdk_json_dt_typ datatype, unsigned long pValue, unsigned long str);
unsigned char getSize(enum brdk_json_dt_typ datatype);

#endif /* !BRDK_JSON_FUNCS */
```

#### brdkJSON_func.c - Internal functions for library.
```c
#include <brdkJSON_func.h>

unsigned long appendBOOL(char value, unsigned long pDestination, unsigned long position, unsigned long size) {
	if(!value) {
		((char*)pDestination)[position++] = BRDK_STR_ASCII_f;
		((char*)pDestination)[position++] = BRDK_STR_ASCII_a;
		((char*)pDestination)[position++] = BRDK_STR_ASCII_l;
		((char*)pDestination)[position++] = BRDK_STR_ASCII_s;
		((char*)pDestination)[position++] = BRDK_STR_ASCII_e;
		return position;
	}
	else {
		((char*)pDestination)[position++] = BRDK_STR_ASCII_t;
		((char*)pDestination)[position++] = BRDK_STR_ASCII_r;
		((char*)pDestination)[position++] = BRDK_STR_ASCII_u;
		((char*)pDestination)[position++] = BRDK_STR_ASCII_e;
		return position;
	}
}

unsigned long setValue(enum brdk_json_dt_typ datatype, unsigned long pValue, unsigned long str) {
	if(datatype == BRDK_JSON_DINT_TO_DINT || datatype == BRDK_JSON_STRING_TO_DINT) {
		signed long* tmpVal = ((signed long*)pValue);
		*tmpVal = brdkStrAToDint(str,BRDK_STR_CONVERT_DECIMAL);
		return 0;
	}
	else if(datatype == BRDK_JSON_UDINT_TO_UDINT || datatype == BRDK_JSON_STRING_TO_UDINT) {
		unsigned long* tmpVal = ((unsigned long*)pValue);
		*tmpVal = brdkStrAToUdint(str,BRDK_STR_CONVERT_DECIMAL);
		return 0;
	}
	else if(datatype == BRDK_JSON_REAL_TO_REAL || datatype == BRDK_JSON_STRING_TO_REAL) {
		float* tmpVal = ((float*)pValue);
		*tmpVal = brdkStrAToReal(str);
		return 0;
	}
	else if(datatype == BRDK_JSON_BOOL_TO_DINT) {
		signed long* tmpVal = ((signed long*)pValue);
		if(brdkStrLen(str) < 0) *tmpVal = false;
		else if(brdkStrCmp(str, (unsigned long)&"true") == 0) *tmpVal = true;
		else if(brdkStrCmp(str, (unsigned long)&"1") == 0) *tmpVal = true;
		else if(brdkStrCmp(str, (unsigned long)&"false") == 0) *tmpVal = false;
		else if(brdkStrCmp(str, (unsigned long)&"0") == 0) *tmpVal = false;
		else if(brdkStrCmp(str, (unsigned long)&"") == 0) *tmpVal = false;
		else return 1;	/* error illegal character */
	}
	else if(datatype == BRDK_JSON_BOOL_TO_UDINT) {
		unsigned long* tmpVal = ((unsigned long*)pValue);
		if(brdkStrLen(str) < 0) *tmpVal = false;
		else if(brdkStrCmp(str, (unsigned long)&"true") == 0) *tmpVal = true;
		else if(brdkStrCmp(str, (unsigned long)&"1") == 0) *tmpVal = true;
		else if(brdkStrCmp(str, (unsigned long)&"false") == 0) *tmpVal = false;
		else if(brdkStrCmp(str, (unsigned long)&"0") == 0) *tmpVal = false;
		else if(brdkStrCmp(str, (unsigned long)&"") == 0) *tmpVal = false;
		else return 1; 	/* error illegal character */
	}
	else {
		char* tmpVal = ((char*)pValue);
		if(brdkStrLen(str) < 0) *tmpVal = false;
		else if(brdkStrCmp(str, (unsigned long)&"true") == 0) *tmpVal = true;
		else if(brdkStrCmp(str, (unsigned long)&"1") == 0) *tmpVal = true;
		else if(brdkStrCmp(str, (unsigned long)&"false") == 0) *tmpVal = false;
		else if(brdkStrCmp(str, (unsigned long)&"0") == 0) *tmpVal = false;
		else if(brdkStrCmp(str, (unsigned long)&"") == 0) *tmpVal = false;
		else return 1; /* error illegal character */
	}
	return 0;
}

unsigned char getSize(enum brdk_json_dt_typ datatype) {
	switch(datatype) {
		case BRDK_JSON_DINT_TO_DINT: case BRDK_JSON_UDINT_TO_UDINT:
		case BRDK_JSON_STRING_TO_DINT: case BRDK_JSON_STRING_TO_UDINT:
		case BRDK_JSON_BOOL_TO_DINT: case BRDK_JSON_BOOL_TO_UDINT:
		case BRDK_JSON_REAL_TO_REAL: case BRDK_JSON_STRING_TO_REAL:
			return 4;
		default:
			return 1;
	}
}
```

### Library Logical/Libraries/brdkSTR (ANSIC, version 1.11.0) - brdk string handling library. Expands string functionality.
Depends on: astime

#### brdkSTR.fun
```iecst
FUNCTION brdkStrAppendDintToA : DINT (*Appends an DINT to the end of a string. $RETURN=length;Length of the string.*) (*$GROUP=User,$CAT=User,$GROUPICON=User.png,$CATICON=User.png*)
	VAR_INPUT
		value : DINT; (*DINT value to be converted.*)
		pString : UDINT; (*String pointer to source string.*)
		base : USINT; (*0,10 = decimal, 2 = binary, 16 = hex.*)
		position : DINT; (*Append position. Negative numbers will count from end of string.*)
	END_VAR
END_FUNCTION

FUNCTION brdkStrAppendUdintToA : DINT (*Appends an UDINT to the end of a string. $RETURN=length;Length of the string.*) (*$GROUP=User,$CAT=User,$GROUPICON=User.png,$CATICON=User.png*)
	VAR_INPUT
		value : UDINT; (*UDINT value to be converted.*)
		pString : UDINT; (*String pointer to source string.*)
		base : USINT; (*0,10 = decimal, 2 = binary, 16 = hex.*)
		position : DINT; (*Append position. Negative numbers will count from end of string.*)
	END_VAR
END_FUNCTION

FUNCTION brdkStrAToDint : DINT (*Converts a string to a DINT type. $RETURN=value;DINT value.*) (*$GROUP=User,$CAT=User,$GROUPICON=User.png,$CATICON=User.png*)
	VAR_INPUT
		pString : UDINT; (*String pointer to source string.*)
		base : USINT; (*0,10 = decimal, 2 = binary, 16 = hex.*)
	END_VAR
END_FUNCTION

FUNCTION brdkStrAToDTStructure : DINT (*Converts a STRING of format yyyy-mm-dd hh:mm:ss.ms into a DTStructure. $RETURN=length;Length of the string.*) (*$GROUP=User,$CAT=User,$GROUPICON=User.png,$CATICON=User.png*)
	VAR_INPUT
		pString : UDINT; (*String pointer to source string.*)
		pDTStructure : UDINT; (*Pointer to the DTStructure.*)
	END_VAR
END_FUNCTION

FUNCTION brdkStrAToReal : REAL (*Converts a string to a REAL type. NB. Implementation not equal to atof(). $RETURN=value;REAL value.*) (*$GROUP=User,$CAT=User,$GROUPICON=User.png,$CATICON=User.png*)
	VAR_INPUT
		pString : UDINT; (*String pointer to source string.*)
	END_VAR
END_FUNCTION

FUNCTION brdkStrAToUdint : UDINT (*Converts a string to an UDINT type. $RETURN=value;UDINT value.*) (*$GROUP=User,$CAT=User,$GROUPICON=User.png,$CATICON=User.png*)
	VAR_INPUT
		pString : UDINT; (*String pointer to source string.*)
		base : USINT; (*0,10 = decimal, 2 = binary, 16 = hex.*)
	END_VAR
END_FUNCTION

FUNCTION brdkStrCat : UDINT (*Appends a copy of the source string to the end of the destination string. $RETURN=address;Address after the string.*) (*$GROUP=User,$CAT=User,$GROUPICON=User.png,$CATICON=User.png*)
	VAR_INPUT
		pDestination : UDINT; (*Destination string pointer.*)
		pSource : UDINT; (*Source string pointer.*)
	END_VAR
END_FUNCTION

FUNCTION brdkStrCatAtChar : DINT (*Appends a copy of the source string to the char position of the destination string. $RETURN=index;Index in destination string where the source string is appended. -1 if char is not found.*) (*$GROUP=User,$CAT=User,$GROUPICON=User.png,$CATICON=User.png*)
	VAR_INPUT
		pDestination : UDINT; (*Destination string pointer.*)
		pSource : UDINT; (*Source string pointer.*)
		pChar : UDINT; (*Char pointer.*)
		direction : DINT; (*0 = first appearance of char, -1 = last appearance of char.*)
		greedy : BOOL; (*If true the source string is appended to the char position. If false the char is still present in the destination string.*)
	END_VAR
END_FUNCTION

FUNCTION brdkStrCharAt : USINT (*Returns the character at the specified index. $RETURN=coding;ASCII coding of the char.*) (*$GROUP=User,$CAT=User,$GROUPICON=User.png,$CATICON=User.png*)
	VAR_INPUT
		pString : UDINT; (*String pointer to source string.*)
		index : UDINT; (*Look up index.*)
		pChar : UDINT; (*Char pointer to char to look up.*)
	END_VAR
END_FUNCTION

FUNCTION brdkStrCharCount : DINT (*Finds how many times a character appears in a string. $RETURN=count;Char count. -1 if error.*) (*$GROUP=User,$CAT=User,$GROUPICON=User.png,$CATICON=User.png*)
	VAR_INPUT
		pString : UDINT; (*String pointer to source string.*)
		pChar : UDINT; (*Pointer to search char.*)
	END_VAR
END_FUNCTION

FUNCTION brdkStrCmp : DINT (*Compares character(s) from string1 to string2. $RETURN=result;0 means that the two string are equal.*)
	VAR_INPUT
		pString1 : UDINT; (*String1 pointer.*)
		pString2 : UDINT; (*String2 pointer.*)
	END_VAR
END_FUNCTION

FUNCTION brdkStrCpy : UDINT (*Copies a string to another string. $RETURN=address;Address after the string.*) (*$GROUP=User,$CAT=User,$GROUPICON=User.png,$CATICON=User.png*)
	VAR_INPUT
		pDestination : UDINT; (*Destination string pointer.*)
		pSource : UDINT; (*Source string pointer.*)
	END_VAR
END_FUNCTION

FUNCTION brdkStrCrc32 : UDINT (*Calculates a CRC32 checksum based on the input string. $RETURN=checksum;Checksum of the string.*) (*$GROUP=User,$CAT=User,$GROUPICON=User.png,$CATICON=User.png*)
	VAR_INPUT
		pString : UDINT; (*String pointer.*)
	END_VAR
END_FUNCTION

FUNCTION brdkStrDintLen : DINT (*Returns the number of characters the DINT value would fill in a STRING. $RETURN=length;string length of the DINT*) (*$GROUP=User,$CAT=User,$GROUPICON=User.png,$CATICON=User.png*)
	VAR_INPUT
		value : DINT; (*DINT value.*)
	END_VAR
END_FUNCTION

FUNCTION brdkStrDintToA : DINT (*Converts a DINT into a STRING type. $RETURN=length;Length of the string.*) (*$GROUP=User,$CAT=User,$GROUPICON=User.png,$CATICON=User.png*)
	VAR_INPUT
		value : DINT; (*DINT value to be converted.*)
		pString : UDINT; (*String pointer to source string.*)
		base : USINT; (*0,10 = decimal, 2 = binary, 16 = hex.*)
	END_VAR
END_FUNCTION

FUNCTION brdkStrDTStructureToA : DINT (*Converts a DTStructure into a STRING type in format yyyy-mm-dd hh:mm:ss.ms. $RETURN=length;Length of the string.*) (*$GROUP=User,$CAT=User,$GROUPICON=User.png,$CATICON=User.png*)
	VAR_INPUT
		pDTStructure : UDINT; (*Pointer to the DTStructure.*)
		pString : UDINT; (*String pointer to destination string.*)
		format : USINT; (*0 = 2020-01-01 01:01:01.001, 1 = 2020-01-01 01:01:01, 2 = 2020-01-01, 3 = 01:01:01, 4 = 01:01:01.001*)
	END_VAR
END_FUNCTION

FUNCTION brdkStrEncode : DINT (*Encodes a string into different formats. $RETURN=address;Address after the string.*) (*$GROUP=User,$CAT=User,$GROUPICON=User.png,$CATICON=User.png*)
	VAR_INPUT
		pDestination : UDINT; (*Destination string pointer.*)
		pSource : UDINT; (*Source string pointer.*)
		format : USINT; (*0 = UTF-8*)
	END_VAR
END_FUNCTION

FUNCTION brdkStrFill : DINT (*Inserts amount of character(s) to the specified position of the string. $RETURN=length;Length of the string. -1 if error.*) (*$GROUP=User,$CAT=User,$GROUPICON=User.png,$CATICON=User.png*)
	VAR_INPUT
		pString : UDINT; (*String pointer to source string.*)
		amount : DINT; (*Fill char amount.*)
		pChar : UDINT; (*Fill char. If 0 whitespace is used.*)
		position : DINT; (*Fill position. Negative numbers will count from end of string.*)
	END_VAR
END_FUNCTION

FUNCTION brdkStrFillUp : DINT (*Fills x amount of character(s) to the specified position of the string. $RETURN=amount;Amount of chars filled. -1 if error.*) (*$GROUP=User,$CAT=User,$GROUPICON=User.png,$CATICON=User.png*)
	VAR_INPUT
		pString : UDINT; (*String pointer to source string.*)
		maxLength : DINT; (*Maximum length of the string.*)
		pChar : UDINT; (*Fill char. If 0 whitespace is used.*)
		position : DINT; (*Fill position. Negative numbers will count from end of string.*)
	END_VAR
END_FUNCTION

FUNCTION brdkStrIndexOf : DINT (*Returns the index within this string of the first or last occurrence of the specified character. $RETURN=index;Index of the char. -1 if char is not found.*) (*$GROUP=User,$CAT=User,$GROUPICON=User.png,$CATICON=User.png*)
	VAR_INPUT
		pString : UDINT; (*String pointer to source string.*)
		pChar : UDINT; (*Char pointer to char to look up.*)
		direction : DINT; (*0 = search from left, -1 = search from right.*)
	END_VAR
END_FUNCTION

FUNCTION brdkStrInsertAtPos : DINT (*Inserts a string into another string at a specified position. $RETURN=length;Length of the string. -1 if error.*) (*$GROUP=User,$CAT=User,$GROUPICON=User.png,$CATICON=User.png*)
	VAR_INPUT
		pString : UDINT; (*String pointer to source string.*)
		pInsert : UDINT; (*String pointer to insert string.*)
		position : DINT; (*Insert position. Negative numbers will count from end of string.*)
	END_VAR
END_FUNCTION

FUNCTION brdkStrIsAlphabet : BOOL (*Returns false or true depending of all characters are present in the alphabet. $RETURN=false/true; a..z = true.*) (*$GROUP=User,$CAT=User,$GROUPICON=User.png,$CATICON=User.png*)
	VAR_INPUT
		pString : UDINT; (*String pointer.*)
	END_VAR
END_FUNCTION

FUNCTION brdkStrIsDigit : BOOL (*Returns false or true depending of all characters are digits. $RETURN=false/true; 0..9 = true.*) (*$GROUP=User,$CAT=User,$GROUPICON=User.png,$CATICON=User.png*)
	VAR_INPUT
		pString : UDINT; (*String pointer.*)
	END_VAR
END_FUNCTION

FUNCTION brdkStrIsEmpty : BOOL (*Returns false or true depending of characters are present in the first position of the string. $RETURN=false/true;Position [0] = /0 = false. Position [0] != /0 = true.*) (*$GROUP=User,$CAT=User,$GROUPICON=User.png,$CATICON=User.png*)
	VAR_INPUT
		pString : UDINT; (*String pointer.*)
	END_VAR
END_FUNCTION

FUNCTION brdkStrJoin : DINT (*Joins elements from a string array into a string with a delimiter. $RETURN=length;Length of the string or error codes.*) (*$GROUP=User,$CAT=User,$GROUPICON=User.png,$CATICON=User.png*)
	VAR_INPUT
		pString : UDINT; (*String pointer to destination string.*)
		pArray : UDINT; (*Pointer to source string array.*)
		pDelimiter : UDINT; (*Delimiter char. If 0 whitespace is used. The delimiter can only be 1 char long.*)
		sizeOfArray : UDINT; (*Max. size of the string array. Size means number of elements in array.*)
		sizeOfArrayString : UDINT; (*Max. size of strings in the array.*)
		sizeOfString : UDINT; (*Max. size of destination string.*)
	END_VAR
END_FUNCTION

FUNCTION brdkStrLen : DINT (*Returns the number of characters in a string. Stops at \0. $RETURN=length;length of the string*) (*$GROUP=User,$CAT=User,$GROUPICON=User.png,$CATICON=User.png*)
	VAR_INPUT
		pString : UDINT; (*String pointer.*)
	END_VAR
END_FUNCTION

FUNCTION brdkStrMemClear : UDINT (*Fills amount of 0 to destination. $RETURN=address;Address after the destination.*) (*$GROUP=User,$CAT=User,$GROUPICON=User.png,$CATICON=User.png*)
	VAR_INPUT
		pDestination : UDINT; (*Destination pointer.*)
		amount : UDINT; (*Amount of character(s) to be initialized.*)
	END_VAR
END_FUNCTION

FUNCTION brdkStrMemCmp : DINT (*Compares amount of character(s) from area1 to area2. $RETURN=result;0 means that the two areas are equal.*) (*$GROUP=User,$CAT=User,$GROUPICON=User.png,$CATICON=User.png*)
	VAR_INPUT
		pArea1 : UDINT; (*Area1 pointer.*)
		pArea2 : UDINT; (*Area2 pointer.*)
		amount : UDINT; (*Amount of character(s) to be comared.*)
	END_VAR
END_FUNCTION

FUNCTION brdkStrMemCpy : UDINT (*Copies amount of character(s) from source to destination. $RETURN=address;Address after the destination.*) (*$GROUP=User,$CAT=User,$GROUPICON=User.png,$CATICON=User.png*)
	VAR_INPUT
		pDestination : UDINT; (*Destination pointer.*)
		pSource : UDINT; (*Source pointer.*)
		amount : UDINT; (*Amount of character(s) to be copied.*)
	END_VAR
END_FUNCTION

FUNCTION brdkStrMemMove : UDINT (*Moves amount of character(s) from source to destination. $RETURN=address;Address after the destination.*) (*$GROUP=User,$CAT=User,$GROUPICON=User.png,$CATICON=User.png*)
	VAR_INPUT
		pDestination : UDINT; (*Destination pointer.*)
		pSource : UDINT; (*Source pointer.*)
		amount : UDINT; (*Amount of character(s) to be moved.*)
	END_VAR
END_FUNCTION

FUNCTION brdkStrMemSet : UDINT (*Fills amount of character(s) to destination. $RETURN=address;Address after the destination.*) (*$GROUP=User,$CAT=User,$GROUPICON=User.png,$CATICON=User.png*)
	VAR_INPUT
		pDestination : UDINT; (*Destination pointer.*)
		value : USINT; (*Initialization value.*)
		amount : UDINT; (*Amount of character(s) to be initialized.*)
	END_VAR
END_FUNCTION

FUNCTION brdkStrMove : UDINT (*Moves a string to another string. $RETURN=address;Address after the string.*) (*$GROUP=User,$CAT=User,$GROUPICON=User.png,$CATICON=User.png*)
	VAR_INPUT
		pDestination : UDINT; (*Destination string pointer.*)
		pSource : UDINT; (*Source string pointer.*)
	END_VAR
END_FUNCTION

FUNCTION brdkStrNAToDint : DINT (*Converts a string to an DINT type for amount of characters. If the function encounters a null character in the source string, if will stop. $RETURN=value;DINT value.*) (*$GROUP=User,$CAT=User,$GROUPICON=User.png,$CATICON=User.png*)
	VAR_INPUT
		pString : UDINT; (*String pointer to source string.*)
		amount : UDINT; (*Amount of character(s) to be converted.*)
		base : USINT; (*0,10 = decimal, 2 = binary, 16 = hex.*)
	END_VAR
END_FUNCTION

FUNCTION brdkStrNAToUdint : UDINT (*Converts a string to an UDINT type for amount of characters. If the function encounters a null character in the source string, if will stop. $RETURN=value;UDINT value.*) (*$GROUP=User,$CAT=User,$GROUPICON=User.png,$CATICON=User.png*)
	VAR_INPUT
		pString : UDINT; (*String pointer to source string.*)
		amount : UDINT; (*Amount of character(s) to be converted.*)
		base : USINT; (*0,10 = decimal, 2 = binary, 16 = hex.*)
	END_VAR
END_FUNCTION

FUNCTION brdkStrNCpy : UDINT (*Copies a string to another string. If the function encounters a null character in the source string, the function will add null characters to the destination string until amount character(s) have been written. $RETURN=address;Address after the string.*) (*$GROUP=User,$CAT=User,$GROUPICON=User.png,$CATICON=User.png*)
	VAR_INPUT
		pDestination : UDINT; (*Destination string pointer.*)
		pSource : UDINT; (*Source string pointer.*)
		amount : UDINT; (*Amount of character(s) to be moved.*)
	END_VAR
END_FUNCTION

FUNCTION brdkStrNIsAlphabet : BOOL (*Returns false or true depending of the amount of characters are present in the alphabet. $RETURN=false/true; a..z = true.*) (*$GROUP=User,$CAT=User,$GROUPICON=User.png,$CATICON=User.png*)
	VAR_INPUT
		pString : UDINT; (*String pointer.*)
		amount : UDINT; (*Amount of character(s) to be checked.*)
	END_VAR
END_FUNCTION

FUNCTION brdkStrNIsDigit : BOOL (*Returns false or true depending of the amount characters are digits. $RETURN=false/true; 0..9 = true.*) (*$GROUP=User,$CAT=User,$GROUPICON=User.png,$CATICON=User.png*)
	VAR_INPUT
		pString : UDINT; (*String pointer.*)
		amount : UDINT; (*Amount of character(s) to be checked.*)
	END_VAR
END_FUNCTION

FUNCTION brdkStrRealToA : DINT (*Converts a REAL into a STRING type. NB. Implementation not equal to ftoa(). $RETURN=length;Length of the string.*) (*$GROUP=User,$CAT=User,$GROUPICON=User.png,$CATICON=User.png*)
	VAR_INPUT
		value : REAL; (*REAL value to be converted.*)
		pString : UDINT; (*String pointer to source string.*)
		precision : USINT; (*Precision of the conversion. Maximum is 10.*)
	END_VAR
END_FUNCTION

FUNCTION brdkStrRemove : UDINT (*Removes character(s) from a string from a specified position. $RETURN=address;Address after the string.*) (*$GROUP=User,$CAT=User,$GROUPICON=User.png,$CATICON=User.png*)
	VAR_INPUT
		pString : UDINT; (*Source string pointer.*)
		start : DINT; (*Index of where to start in the string. Negative numbers start from the end of the string.*)
		length : DINT; (*0 means to the end of the string. Negative length is subtracted from the end of the string. Is start is negative length is subtracted from the start of the string. *)
	END_VAR
END_FUNCTION

FUNCTION brdkStrRepeat : DINT (*Repeats a string a specified number of times. $RETURN=length;Length of the string.*) (*$GROUP=User,$CAT=User,$GROUPICON=User.png,$CATICON=User.png*)
	VAR_INPUT
		pString : UDINT; (*String pointer to source string.*)
		times : DINT; (*Number of times the string should be repeated.*)
	END_VAR
END_FUNCTION

FUNCTION brdkStrReplace : DINT (*Replaces some characters with some other characters in a string. $RETURN=number;Number of replacements done.*) (*$GROUP=User,$CAT=User,$GROUPICON=User.png,$CATICON=User.png*)
	VAR_INPUT
		pString : UDINT; (*String pointer to source string.*)
		pFind : UDINT; (*String pointer to find string.*)
		pReplace : UDINT; (*String pointer to replacement string:*)
	END_VAR
END_FUNCTION

FUNCTION brdkStrReverse : DINT (*Reverses a string from start position to end position. $RETURN=count;Number of reverses done. -1 if error.*) (*$GROUP=User,$CAT=User,$GROUPICON=User.png,$CATICON=User.png*)
	VAR_INPUT
		pString : UDINT; (*String pointer to source string.*)
		startPosition : DINT; (*Start position. Must be a positive number and less than length.*)
		endPosition : DINT; (*End position. Must be less than length unless it's a negative numbers which will count from end of string.*)
	END_VAR
END_FUNCTION

FUNCTION brdkStrReverseWords : DINT (*Reverses words in a string. $RETURN=count;Number of words reversed.*) (*$GROUP=User,$CAT=User,$GROUPICON=User.png,$CATICON=User.png*)
	VAR_INPUT
		pString : UDINT; (*String pointer to source string.*)
	END_VAR
END_FUNCTION

FUNCTION brdkStrSearch : DINT (*Searches a string for a specified string. $RETURN=position; Position of the match. -1 if no match.*) (*$GROUP=User,$CAT=User,$GROUPICON=User.png,$CATICON=User.png*)
	VAR_INPUT
		pString : UDINT; (*String pointer to source string.*)
		pSearchString : UDINT; (*String pointer to search string.*)
	END_VAR
END_FUNCTION

FUNCTION brdkStrSlice : DINT (*Slices a part of a string. $RETURN=length;Length of the string. -1 if error.*) (*$GROUP=User,$CAT=User,$GROUPICON=User.png,$CATICON=User.png*)
	VAR_INPUT
		pString : UDINT; (*String pointer to source string.*)
		start : DINT; (*Start position.*)
		end : DINT; (*End position.*)
	END_VAR
END_FUNCTION

FUNCTION brdkStrSplit : DINT (*Splits a string into an array of string using a seperator. $RETURN=count;Number of elements splitted or an error code.*) (*$GROUP=User,$CAT=User,$GROUPICON=User.png,$CATICON=User.png*)
	VAR_INPUT
		pArray : UDINT; (*Pointer to destination string array.*)
		pString : UDINT; (*String pointer to source string.*)
		pDelimiter : UDINT; (*Delimiter char. If 0 whitespace is used. The delimiter can only be 1 char long.*)
		sizeOfArray : UDINT; (*Max. size of the string array. Size means number of elements in array.*)
		sizeofArrayString : UDINT; (*Max. size of strings in the array.*)
		greedy : BOOL; (*Remove or keep the seperator from the string.*)
	END_VAR
END_FUNCTION

FUNCTION brdkStrSubDintSearch : DINT (*Returns a DINT based on a search. $RETURN=length;Length of the destination string. -1 if error.*) (*$GROUP=User,$CAT=User,$GROUPICON=User.png,$CATICON=User.png*)
	VAR_INPUT
		pSource : UDINT; (*Source string pointer.*)
		pStart : UDINT; (*String pointer for start search string.*)
		pEnd : UDINT; (*String pointer for end search string. The function will only search after the start string.*)
		startOffset : DINT; (*Offset for the start poition. If greedy = true offset is after the start has been removed.*)
		base : USINT; (*0,10 = decimal, 2 = binary, 16 = hex.*)
	END_VAR
END_FUNCTION

FUNCTION brdkStrSubStr : DINT (*Returns a part of a string. $RETURN=length;Length of the destination string. -1 if error.*) (*$GROUP=User,$CAT=User,$GROUPICON=User.png,$CATICON=User.png*)
	VAR_INPUT
		pDestination : UDINT; (*Destination string pointer.*)
		pSource : UDINT; (*Source string pointer.*)
		start : DINT; (*Index of where to start in the string. Negative numbers start from the end of the string.*)
		length : DINT; (*0 means to the end of the string. Negative length is subtracted from the end of the string. Is start is negative length is subtracted from the start of the string. *)
	END_VAR
END_FUNCTION

FUNCTION brdkStrSubStrSearch : BOOL (*Returns a part of a string based on a search. $RETURN=success;TRUE = success *) (*$GROUP=User,$CAT=User,$GROUPICON=User.png,$CATICON=User.png*)
	VAR_INPUT
		pDestination : UDINT; (*Destination string pointer.*)
		pSource : UDINT; (*Source string pointer.*)
		pStart : UDINT; (*String pointer for start search string.*)
		pEnd : UDINT; (*String pointer for end search string. The function will only search after the start string.*)
		startOffset : DINT; (*Offset for the start poition. If greedy = true offset is after the start has been removed.*)
		greedy : BOOL; (*Will add or remove the search strings from the destination string.*)
	END_VAR
END_FUNCTION

FUNCTION brdkStrToDec : DINT (*Converts a string of hexadecimal values to ASCII characters. $RETURN=length;Length of the string. -1 if error.*) (*$GROUP=User,$CAT=User,$GROUPICON=User.png,$CATICON=User.png*)
	VAR_INPUT
		pString : UDINT; (*String pointer to source string.*)
	END_VAR
END_FUNCTION

FUNCTION brdkStrToHex : DINT (*Converts a string of ASCII characters to hexadecimal values. $RETURN=length;Length of the string.*) (*$GROUP=User,$CAT=User,$GROUPICON=User.png,$CATICON=User.png*)
	VAR_INPUT
		pString : UDINT; (*String pointer to source string.*)
	END_VAR
END_FUNCTION

FUNCTION brdkStrToLowerCase : DINT (*Converts a string to lowercase letters. $RETURN=number;Number of characters changed.*) (*$GROUP=User,$CAT=User,$GROUPICON=User.png,$CATICON=User.png*)
	VAR_INPUT
		pString : UDINT; (*String pointer to source string.*)
	END_VAR
END_FUNCTION

FUNCTION brdkStrToUpperCase : DINT (*Converts a string to uppercase letters. $RETURN=number;Number of characters changed.*) (*$GROUP=User,$CAT=User,$GROUPICON=User.png,$CATICON=User.png*)
	VAR_INPUT
		pString : UDINT; (*String pointer to source string.*)
	END_VAR
END_FUNCTION

FUNCTION brdkStrToUpperCaseWords : DINT (*Convert the first character of each word to uppercase. (title()). $RETURN=number;Number of characters changed.*) (*$GROUP=User,$CAT=User,$GROUPICON=User.png,$CATICON=User.png*)
	VAR_INPUT
		pString : UDINT; (*String pointer to source string.*)
	END_VAR
END_FUNCTION

FUNCTION brdkStrTrim : DINT (*Removes whitespaces from a string. $RETURN=number;Number of whitespaces removed from string.*) (*$GROUP=User,$CAT=User,$GROUPICON=User.png,$CATICON=User.png*)
	VAR_INPUT
		pString : UDINT; (*String pointer to source string.*)
		direction : DINT; (*0 = both sides, 1 = left side only, -1 = right side only.*)
	END_VAR
END_FUNCTION

FUNCTION brdkStrUdintLen : DINT (*Returns the number of characters the UDINT value would fill in a STRING. $RETURN=length;string length of the UDINT*) (*$GROUP=User,$CAT=User,$GROUPICON=User.png,$CATICON=User.png*)
	VAR_INPUT
		value : UDINT; (*UDINT value.*)
	END_VAR
END_FUNCTION

FUNCTION brdkStrUdintToA : DINT (*Converts an UDINT into a STRING type. $RETURN=length;Length of the string.*) (*$GROUP=User,$CAT=User,$GROUPICON=User.png,$CATICON=User.png*)
	VAR_INPUT
		value : UDINT; (*UDINT value to be converted.*)
		pString : UDINT; (*String pointer to source string.*)
		base : USINT; (*0,10 = decimal, 2 = binary, 16 = hex.*)
	END_VAR
END_FUNCTION

FUNCTION brdkStrWord : DINT (*Returns a word in a string given by a number and a delimiter. $RETURN=length;Length of the string.*) (*$GROUP=User,$CAT=User,$GROUPICON=User.png,$CATICON=User.png*)
	VAR_INPUT
		pDestination : UDINT; (*Destination string pointer.*)
		pSource : UDINT; (*Source string pointer.*)
		pDelimiter : UDINT; (*Delimiter char. If 0 whitespace is used. The delimiter can only be 1 char long.*)
		number : DINT; (*Word number in string. 1 = first word. -1 = last word.*)
		sizeOfString : UDINT; (*Max. size of destination string.*)
	END_VAR
END_FUNCTION
```

#### brdkStrAppendDintToA.c
```c
#include <brdkSTR_func.h>

signed long brdkStrAppendDintToA(signed long value, unsigned long pString, unsigned char base, signed long position) {
	signed long start,i,cnt=0;
	if(value < 0) {
		if(position > -1) start = position;
		else start = brdkStrLen(pString);

		brdkStrFill(pString,1,(unsigned long)&"-",start++);
		i = start;
		value *= -1;
		base = !base ? 10 : base;	/* make sure base is not 0 */
		while (value > 0) {
			unsigned long rem = value % base;
			unsigned char tmp = (rem > 9)? (rem-10) + BRDK_STR_ASCII_A : rem + BRDK_STR_ASCII_0;
			brdkStrFill(pString,1,(unsigned long)&tmp,i++);
	       	value = value/base;
			cnt++;
		}
		brdkStrReverse(pString,start,--i);
		if(position < 0) ((char*)pString)[start+cnt] = BRDK_STR_ASCII_NULL;
		return start+cnt+brdkStrLen(pString+start+cnt);
	}
	else return brdkStrAppendUdintToA(value,pString,base,position);
}
```

#### brdkStrAppendUdintToA.c
```c
#include <brdkSTR_func.h>

signed long brdkStrAppendUdintToA(unsigned long value, unsigned long pString, unsigned char base, signed long position) {
	signed long start,i,cnt=0;
	if(position > -1) start = position;
	else start = brdkStrLen(pString);
	i = start;
	if (value != 0) {
		base = !base ? 10 : base;	/* make sure base is not 0 */
		while (value > 0) {
			unsigned long rem = value % base;
			unsigned char tmp = (rem > 9)? (rem-10) + BRDK_STR_ASCII_A : rem + BRDK_STR_ASCII_0;
			brdkStrFill(pString,1,(unsigned long)&tmp,i++);
	       	value = value/base;
			cnt++;
		}
		brdkStrReverse(pString,start,--i);
		if(position < 0) ((char*)pString)[start+cnt] = BRDK_STR_ASCII_NULL;
		return start+cnt+brdkStrLen(pString+start+cnt);
	}
	else {
		((char*)pString)[start++] = BRDK_STR_ASCII_0;
		((char*)pString)[start] = BRDK_STR_ASCII_NULL;
		return start;
	}
}
```

#### brdkStrAToReal.c
```c
#include <brdkSTR_func.h>

float brdkStrAToReal(unsigned long pString) {
	float value = 0.0, fraction = 0.1;
	signed long exponent = 0;
	unsigned char sign = 0;
	unsigned long i = 0;

	while (((char*)pString)[i] == BRDK_STR_ASCII_SPACE || ((char*)pString)[i] == BRDK_STR_ASCII_PLUS) i++;	/* Remove white spaces or + sign */
	if(((char*)pString)[i] == BRDK_STR_ASCII_HYPHEN) {
		sign = 1;
		i++;
	}
	/* integer section */
	while(isDigit(((char*)pString)[i])) {
		value = (value * 10.0) + (((char*)pString)[i]-BRDK_STR_ASCII_0);
		i++;
	}
	/* fraction section */
	if((((char*)pString)[i]) == BRDK_STR_ASCII_DOT) {
		i++;
		while(isDigit(((char*)pString)[i])) {
			value += (((char*)pString)[i]-BRDK_STR_ASCII_0) * fraction;
			fraction *= 0.1;
			i++;
		}
	}
	/* exponent section */
	if((((char*)pString)[i]) == BRDK_STR_ASCII_E || (((char*)pString)[i]) == BRDK_STR_ASCII_e) {
		i++;
		exponent = brdkStrAToDint(pString+i,BRDK_STR_CONVERT_DECIMAL);
		while(exponent != 0) {
			if(exponent < 0) {
				value *= 0.1;
				exponent++;
			}
			else {
				value *= 10.0;
				exponent--;
			}
		}
	}

	if(sign) value *= -1.0;
	return (value);
}
```

#### brdkStrDintLen.c
```c
#include <brdkSTR_func.h>

signed long brdkStrDintLen(signed long value) {
	if(value < 10 && value > -10) return 1 + (value < 0);
	else if(value < 100 && value > -100) return 2 + (value < 0);
	else if(value < 1000 && value > -1000) return 3 + (value < 0);
	else if(value < 10000 && value > -10000) return 4 + (value < 0);
	else if(value < 100000 && value > -100000) return 5 + (value < 0);
	else if(value < 1000000 && value > -1000000) return 6 + (value < 0);
	else if(value < 10000000 && value > -10000000) return 7 + (value < 0);
	else if(value < 100000000 && value > -100000000) return 8 + (value < 0);
	else if(value < 1000000000 && value > -1000000000) return 9 + (value < 0);
	else return 10;
}
```

#### brdkStrDTStructureToA.c
```c
#include <brdkSTR_func.h>

signed long brdkStrDTStructureToA(unsigned long pDTStructure, unsigned long pString, unsigned char format) {
	/* format 0 = 2020-01-01 01:01:01.001 */
	/* format 1 = 2020-01-01 01:01:01 */
	/* format 2 = 2020-01-01 */
	/* format 3 = 01:01:01 */
	/* format 4 = 01:01:01.001 */
	DTStructure* dtStruct = (DTStructure*)pDTStructure;
	unsigned char pos = 0;
	if(format != 3 && format != 4) {
		brdkStrUdintToA(dtStruct->year,(unsigned long)&(((char*)pString)[0]),BRDK_STR_CONVERT_DECIMAL);
		((char*)pString)[4] = BRDK_STR_ASCII_HYPHEN;
		if(dtStruct->month < 10) {
			((char*)pString)[5] = BRDK_STR_ASCII_0;
			brdkStrUdintToA(dtStruct->month,(unsigned long)&(((char*)pString)[6]),BRDK_STR_CONVERT_DECIMAL);
		}
		else brdkStrUdintToA(dtStruct->month,(unsigned long)&(((char*)pString)[5]),BRDK_STR_CONVERT_DECIMAL);
		((char*)pString)[7] = BRDK_STR_ASCII_HYPHEN;
		if(dtStruct->day < 10) {
			((char*)pString)[8] = BRDK_STR_ASCII_0;
			brdkStrUdintToA(dtStruct->day,(unsigned long)&(((char*)pString)[9]),BRDK_STR_CONVERT_DECIMAL);
		}
		else brdkStrUdintToA(dtStruct->day,(unsigned long)&(((char*)pString)[8]),BRDK_STR_CONVERT_DECIMAL);
		if(format == 2) {
			((char*)pString)[10] = BRDK_STR_ASCII_NULL;
			return 10;
		}
		((char*)pString)[10] = BRDK_STR_ASCII_SPACE;
		pos = 11;
	}
	if(dtStruct->hour < 10) {
		((char*)pString)[pos++] = BRDK_STR_ASCII_0;
		brdkStrUdintToA(dtStruct->hour,(unsigned long)&(((char*)pString)[pos++]),BRDK_STR_CONVERT_DECIMAL);
	}
	else {
		brdkStrUdintToA(dtStruct->hour,(unsigned long)&(((char*)pString)[pos++]),BRDK_STR_CONVERT_DECIMAL);
		pos++;
	}
	((char*)pString)[pos++] = BRDK_STR_ASCII_COLON;
	if(dtStruct->minute < 10) {
		((char*)pString)[pos++] = BRDK_STR_ASCII_0;
		brdkStrUdintToA(dtStruct->minute,(unsigned long)&(((char*)pString)[pos++]),BRDK_STR_CONVERT_DECIMAL);
	}
	else {
		brdkStrUdintToA(dtStruct->minute,(unsigned long)&(((char*)pString)[pos++]),BRDK_STR_CONVERT_DECIMAL);
		pos++;
	}
	((char*)pString)[pos++] = BRDK_STR_ASCII_COLON;
	if(dtStruct->second < 10) {
		((char*)pString)[pos++] = BRDK_STR_ASCII_0;
		brdkStrUdintToA(dtStruct->second,(unsigned long)&(((char*)pString)[pos++]),BRDK_STR_CONVERT_DECIMAL);
	}
	else {
		brdkStrUdintToA(dtStruct->second,(unsigned long)&(((char*)pString)[pos++]),BRDK_STR_CONVERT_DECIMAL);
		pos++;
	}
	if(format == 1 || format == 3) {
		((char*)pString)[pos] = BRDK_STR_ASCII_NULL;
		return pos;
	}
	((char*)pString)[pos++] = BRDK_STR_ASCII_DOT;
	if(dtStruct->millisec < 10) {
		((char*)pString)[pos++] = BRDK_STR_ASCII_0;
		((char*)pString)[pos++] = BRDK_STR_ASCII_0;
		brdkStrUdintToA(dtStruct->millisec,(unsigned long)&(((char*)pString)[pos++]),BRDK_STR_CONVERT_DECIMAL);
	}
	else if(dtStruct->millisec < 100) {
		((char*)pString)[pos++] = BRDK_STR_ASCII_0;
		brdkStrUdintToA(dtStruct->millisec,(unsigned long)&(((char*)pString)[pos++]),BRDK_STR_CONVERT_DECIMAL);
		pos++;
	}
	else {
		brdkStrUdintToA(dtStruct->millisec,(unsigned long)&(((char*)pString)[pos++]),BRDK_STR_CONVERT_DECIMAL);
		pos += 2;
	}
	if(format == 4) {
		((char*)pString)[pos] = BRDK_STR_ASCII_NULL;
		return pos;
	}
	((char*)pString)[pos] = BRDK_STR_ASCII_NULL;
	return pos;
}
```

#### brdkStrIsAlphabet.c
```c
#include <brdkSTR_func.h>

unsigned char brdkStrIsAlphabet(unsigned long pString) {
	unsigned long len = 0;
	while(((char*)pString)[len]) if(!isAlphabet(((char*)pString)[len++])) return 0;
	return 1;
}
```

#### brdkStrIsDigit.c
```c
#include <brdkSTR_func.h>

unsigned char brdkStrIsDigit(unsigned long pString) {
	unsigned long len = 0;
	while(((char*)pString)[len]) if(!isDigit(((char*)pString)[len++])) return 0;
	return 1;
}
```

#### brdkStrNAToUdint.c
```c
#include <brdkSTR_func.h>

unsigned long brdkStrNAToUdint(unsigned long pString, unsigned long amount, unsigned char base) {
	unsigned long value = 0,i;
	if(amount > 0) {
		for(i=0; i < amount; i++) {
			switch(base) {

				case 0: case 10:
					if(isDigit(((char*)pString)[i])) value = (value * 10) + (((char*)pString)[i]-BRDK_STR_ASCII_0);
					else {
						value = 0;
						i = amount;
					}
					break;

				case 2:
					if(((char*)pString)[i] >= BRDK_STR_ASCII_0 && ((char*)pString)[i] <= BRDK_STR_ASCII_1) value += (((char*)pString)[i]-BRDK_STR_ASCII_0)*(1<<(amount-1-i));			/* 0x30 = 0, 0x31 = 1 */
					else {
						value = 0;
						i = amount;
					}
					break;

				case 16:
					if(isDigit(((char*)pString)[i])) 	value += (((char*)pString)[i]-BRDK_STR_ASCII_0)*(1<<(4*(amount-1-i)));		/* 0x30 = 0, 0x39 = 9 */
					else if(((char*)pString)[i] >= BRDK_STR_ASCII_A && ((char*)pString)[i] <= BRDK_STR_ASCII_F) value += (((char*)pString)[i]-BRDK_STR_ASCII_7)*(1<<(4*(amount-1-i)));	/* 0x41 = A, 0x46 = F */
					else if(((char*)pString)[i] >= BRDK_STR_ASCII_a && ((char*)pString)[i] <= BRDK_STR_ASCII_f)value += (((char*)pString)[i]-BRDK_STR_ASCII_W)*(1<<(4*(amount-1-i)));	/* 0x61 = a, 0x66 = f */
					else {
						value = 0;
						i = amount;
					}
					break;

				default:
					value = 0;
					i = amount;
					break;

			}
		}
	}
	return value;
}
```

#### brdkStrNIsAlphabet.c
```c
#include <brdkSTR_func.h>

unsigned char brdkStrNIsAlphabet(unsigned long pString, unsigned long amount) {
	unsigned long len = 0;
	while(len < amount) if(!isAlphabet(((char*)pString)[len++])) return 0;
	return 1;
}
```

#### brdkStrNIsDigit.c
```c
#include <brdkSTR_func.h>

unsigned char brdkStrNIsDigit(unsigned long pString, unsigned long amount) {
	unsigned long len = 0;
	while(len < amount) if(!isDigit(((char*)pString)[len++])) return 0;
	return 1;
}
```

#### brdkStrRealToA.c
```c
#include <brdkSTR_func.h>

static const float rounds[] = {
	0.5,
	0.05,
	0.005,
	0.0005,
	0.00005,
	0.000005,
	0.0000005,
	0.00000005,
	0.000000005,
	0.0000000005,
	0.00000000005
};

signed long brdkStrRealToA(float value, unsigned long pString, unsigned char precision) {
	signed long i = 0;
	char tmpChar;
	unsigned long integer;
	if(precision > 10) precision = 10;
	if (value < 0) {
		value = -value;
		((char*)pString)[i++] = BRDK_STR_ASCII_HYPHEN;
	}

	if(precision) value += rounds[precision];

	/* handle integer section */
	integer = value;
	value -= integer;

	if(integer > 0) i += brdkStrUdintToA(integer,pString+i,BRDK_STR_CONVERT_DECIMAL);
	else ((char*)pString)[i++] = BRDK_STR_ASCII_0;

	/* handle decimal section */
	if(precision) {
		((char*)pString)[i++] = BRDK_STR_ASCII_DOT;

		while(precision--) {
			value *= 10.0;
			tmpChar = value;
			((char*)pString)[i++] = BRDK_STR_ASCII_0 + tmpChar;
			value -= tmpChar;
		}
	}

	((char*)pString)[i] = BRDK_STR_ASCII_NULL;
	return i;
}
```

#### brdkStrUdintLen.c
```c
#include <brdkSTR_func.h>

signed long brdkStrUdintLen(unsigned long value) {
	if(value < 10) return 1;
	else if(value < 100) return 2;
	else if(value < 1000) return 3;
	else if(value < 10000) return 4;
	else if(value < 100000) return 5;
	else if(value < 1000000) return 6;
	else if(value < 10000000) return 7;
	else if(value < 100000000) return 8;
	else if(value < 1000000000) return 9;
	else return 10;
}
```

#### brdkStrUdintToA.c
```c
#include <brdkSTR_func.h>

signed long brdkStrUdintToA(unsigned long value, unsigned long pString, unsigned char base) {
	signed long len = 0;
	if (value != 0) {
		((char*)pString)[0] = 0;
		base = !base ? 10 : base;	/* make sure base is not 0 */
		while (value > 0) {
			unsigned long rem = value % base;
	       	((char*)pString)[len++] = (rem > 9)? (rem-10) + BRDK_STR_ASCII_A : rem + BRDK_STR_ASCII_0;
	       	value = value/base;
		}
		((char*)pString)[len] = BRDK_STR_ASCII_NULL;
		brdkStrReverse(pString,0,-1);
	}
	else {
		((char*)pString)[0] = BRDK_STR_ASCII_0;
		((char*)pString)[1] = BRDK_STR_ASCII_NULL;
		len = 1;
	}
	return len;
}
```

#### brdkSTR_func.h
```c
#ifndef BRDK_STR_FUNCS
#define BRDK_STR_FUNCS 1

#include <brdkSTR.h>
#include <bur/plctypes.h>

#ifdef __cplusplus
	extern "C"
	{
#endif

signed long search(signed long pString, signed long lenString, signed long pSearchString, signed long lenSearch);
unsigned char dayOfWeek(unsigned char d,unsigned char m, unsigned short y);
unsigned char isDigit(char c);
unsigned char isAlphabet(char c);
float strtof(char *string, char **endPtr);

#ifdef __cplusplus
	};
#endif

#endif
```

#### brdkSTR_func.c
```c
#include <brdkSTR_func.h>

/* search for a string in a string */
signed long search(signed long pString, signed long lenString, signed long pSearchString, signed long lenSearch) {
	signed long pos=-1, i=0,j=0;
	if(lenString>=lenSearch) {
		for(i=0; i <= lenString-lenSearch; i++) {
			j=0;
			if(((char*)pString)[i] == ((char*)pSearchString)[j]) {
				while(((char*)pString)[i+j] == ((char*)pSearchString)[j]) {
					j++;
					if(j==lenSearch) {
						pos = i;
						i=lenString-lenSearch+1;
						break;
					}
				}
			}
		}
	}
	return pos;
}

unsigned char dayOfWeek(unsigned char d,unsigned char m, unsigned short y){
	unsigned char t[] = { 0, 3, 2, 5, 0, 3, 5, 1, 4, 6, 2, 4 };
	if (m < 3) y -= 1;
	return((y + y / 4 - y / 100 + y / 400 + t[m - 1] + d) % 7);
}

/* 0x30 = 0, 0x39 = 9 */
unsigned char isDigit(char c) {
	return ((c >= BRDK_STR_ASCII_0) && (c <= BRDK_STR_ASCII_9));
}

unsigned char isAlphabet(char c) {
	return (((c >= BRDK_STR_ASCII_A) && (c <= BRDK_STR_ASCII_Z))) || (((c >= BRDK_STR_ASCII_a) && (c <= BRDK_STR_ASCII_z)));
}
```

- CHANGELOG - brdkSTR change log (not shown)

### Library Logical/Libraries/Goertzel (IEC)

#### freqHelp.var - Exported constants
```iecst
VAR CONSTANT
	MAX_SAMPLES_GOERTZEL : UINT := 100;
END_VAR
```

#### Goertzel.fun - Exported functions and function blocks
```iecst
FUNCTION goertzel : REAL
	VAR_INPUT
		samples : REFERENCE TO ARRAY[0..MAX_SAMPLES_GOERTZEL] OF REAL;
		frequency : REAL;
		sampleRate : UINT;
	END_VAR
	VAR
		r : REAL;
		w : REAL;
		cosine : REAL;
		sine : REAL;
		coeff : REAL;
		Q0 : REAL;
		Q1 : REAL;
		Q2 : REAL;
		j : UINT;
		real : REAL;
		imag : REAL;
	END_VAR
END_FUNCTION

FUNCTION goertzelWindowSmooth : REAL
	VAR_INPUT
		samples : REFERENCE TO ARRAY[0..MAX_SAMPLES_GOERTZEL] OF REAL;
		window : REFERENCE TO ARRAY[0..MAX_SAMPLES_GOERTZEL] OF REAL;
		frequency : REAL;
		sampleRate : UINT;
	END_VAR
	VAR
		r : REAL;
		w : REAL;
		cosine : REAL;
		sine : REAL;
		coeff : REAL;
		Q0 : REAL;
		Q1 : REAL;
		Q2 : REAL;
		j : UINT;
		real : REAL;
		imag : REAL;
	END_VAR
END_FUNCTION

FUNCTION getHammingWindow : REAL
	VAR_INPUT
		N : REAL;
		n : REAL;
	END_VAR
END_FUNCTION

FUNCTION_BLOCK goertzelMagPhase
	VAR_INPUT
		samples : REFERENCE TO ARRAY[0..MAX_SAMPLES_GOERTZEL] OF REAL;
		window : REFERENCE TO ARRAY[0..MAX_SAMPLES_GOERTZEL] OF REAL;
		frequency : {REDUND_UNREPLICABLE} REAL;
		sampleRate : {REDUND_UNREPLICABLE} UINT;
	END_VAR
	VAR
		r : {REDUND_UNREPLICABLE} REAL;
		w : {REDUND_UNREPLICABLE} REAL;
		cosine : {REDUND_UNREPLICABLE} REAL;
		sine : {REDUND_UNREPLICABLE} REAL;
		coeff : {REDUND_UNREPLICABLE} REAL;
		Q0 : {REDUND_UNREPLICABLE} REAL;
		Q1 : {REDUND_UNREPLICABLE} REAL;
		Q2 : {REDUND_UNREPLICABLE} REAL;
		j : {REDUND_UNREPLICABLE} UINT;
		real : {REDUND_UNREPLICABLE} REAL;
		imag : {REDUND_UNREPLICABLE} REAL;
	END_VAR
	VAR_OUTPUT
		magnitude  : REAL;
		phase : REAL;
	END_VAR
END_FUNCTION_BLOCK
```

#### goertzel.st
```iecst
(* Implementation of Goertzel algorithm in Structured Text *)
FUNCTION goertzel

	r := (PI*2)/UINT_TO_REAL(sampleRate);

	w := r*frequency;
	cosine := COS(w);
	sine := SIN(w);
	coeff := 2*cosine;
	Q0 := 0;
	Q1 := 0;
	Q2 := 0;

	FOR j:=0 TO MAX_SAMPLES_GOERTZEL DO
		Q0 := coeff * Q1 - Q2 + (samples[j]);
		Q2 := Q1;
		Q1 := Q0;
	END_FOR

	real := Q1 - Q2 * cosine;
	imag := Q2 * sine;

	goertzel := SQRT(((real*real)+(imag*imag)));

END_FUNCTION

FUNCTION goertzelWindowSmooth

	r := (PI*2)/UINT_TO_REAL(sampleRate);

	w := r*frequency;
	cosine := COS(w);
	sine := SIN(w);
	coeff := 2*cosine;
	Q0 := 0;
	Q1 := 0;
	Q2 := 0;

	FOR j:=0 TO MAX_SAMPLES_GOERTZEL DO
		Q0 := coeff * Q1 - Q2 + (samples[j]*window[j]);
		Q2 := Q1;
		Q1 := Q0;
	END_FOR

	real := Q1 - Q2 * cosine;
	imag := Q2 * sine;

	goertzelWindowSmooth := SQRT(((real*real)+(imag*imag)));

END_FUNCTION

FUNCTION_BLOCK goertzelMagPhase

	r := (PI*2)/UINT_TO_REAL(sampleRate);

	w := r*frequency;
	cosine := COS(w);
	sine := SIN(w);
	coeff := 2*cosine;
	Q0 := 0;
	Q1 := 0;
	Q2 := 0;

	FOR j:=0 TO MAX_SAMPLES_GOERTZEL DO
		Q0 := coeff * Q1 - Q2 + (samples[j]*window[j]);
		Q2 := Q1;
		Q1 := Q0;
	END_FOR

	real := Q1 - Q2 * cosine;
	imag := Q2 * sine;

	magnitude := SQRT(((real*real)+(imag*imag)));;
	phase := atan2(imag,real);

END_FUNCTION_BLOCK
```

#### getHammingWindow.st
```iecst
(* Implementation of Goertzel algorithm in Structured Text *)
FUNCTION getHammingWindow

	getHammingWindow := 0.54 - 0.46 * COS(((PI*2) * n)/(N - 1));;

END_FUNCTION
```

- Visualisation Logical/mappView (not shown)

### Program Logical/modules/sampling (IEC)
